// TwinCAT 3 PLC project _2AngleProPLC
// ProgramVersion: 3.1.4024.0
// libraries:
//   Tc2_MC2, * (Beckhoff Automation GmbH)
//   Tc2_Standard, * (Beckhoff Automation GmbH)
//   Tc2_System, * (Beckhoff Automation GmbH)
//   Tc3_Module, * (Beckhoff Automation GmbH)
// project tree:
//   DUTs/ AnalogSignal.TcDUT, SSI_Encoder.TcDUT, ST_IOcard.TcDUT
//   / GlobalTextList.TcGTLO, PlcTask.TcTTO, Visualization Manager.TcVMO (not stored)
//   GVLs/ GVL.TcGVL, GVL_Retain.TcGVL, IO.TcGVL, TwinSAFE.TcGVL
//   POUs/FUNCTION BLOCKS/ FB_AnalogIn.TcPOU, FB_Blinker.TcPOU, FB_IntFilter.TcPOU, FB_SSI_Encoder.TcPOU, InverseAnalogControl.TcPOU
//   POUs/MAIN FUNCTIONS/ PRG_00_General.TcPOU, PRG_01_Reel.TcPOU, PRG_02_Xdrive.TcPOU, PRG_03_Saw.TcPOU, PRG_04_SawAxes.TcPOU, PRG_05_Turret_Carriage.TcPOU, PRG_06_HomePosition.TcPOU, PRG_07_Servo.TcPOU, PRG_08_AnalogSignal.TcPOU, PRG_XX_Visualization_Variables.TcPOU
//   POUs/ MAIN.TcPOU, PRG_IO.TcPOU
//   VISUs/ Visualization.TcVIS
// real-time tasks:
//   TASK PlcTask: cycle T#10ms, priority 20, ADS port 350
// motion (NC):
//   TASK NC-Task 1 SAF: cycle T#2ms, priority 4, ADS port 501
//   TASK NC-Task 1 SVB: cycle T#10ms, priority 8, ADS port 511
//   AXIS Axis 1 (id 1)
//     OtherSettings: AllowMotionCmdToSlave=true
//     encoder EncType=19
//       EncPara: MaxCount=#xffffffff
//     drive DrvType=16
//       DrvPara: MaxCount=#xffffffff, DriveControlDWord=#x00020100
//         Analog: TorqueSetpointScale=10, ScaleFactorActTorque=0.1
//         TimeComp: TaskDelayCycles=1
//     controller CtrType=1
//       CtrPara: PriorControlFactor=1
//         Observer: BandWidth=20
//   AXIS Axis 2 (id 2)
//     OtherSettings: AllowMotionCmdToSlave=true
//     encoder EncType=19
//       EncPara: MaxCount=#xffffffff
//     drive DrvType=16
//       DrvPara: MaxCount=#xffffffff, DriveControlDWord=#x00020100
//         Analog: TorqueSetpointScale=10, ScaleFactorActTorque=0.1
//         TimeComp: TaskDelayCycles=1
//     controller CtrType=1
//       CtrPara: PriorControlFactor=1
//         Observer: BandWidth=20
// I/O:
//   DEVICE Device 1 (EtherCAT), AmsNetId 5.146.75.130.2.1
//     AK1 (EK1200) [EK1200-5000 EtherCAT Power supply (2A E-Bus)]
//       SI1 (EL6910) [EL6910, TwinSAFE PLC]
//       ID1 (EL1018) [EL1018 8Ch. Dig. Input 24V, 10µs]
//       ID2 (EL1018) [EL1018 8Ch. Dig. Input 24V, 10µs]
//       IS1 (EL1904) [EL1904, 4 Ch. Safety Input 24V, TwinSAFE]
//         modules: Module 1 (FSOES)
//       IS2 (EL1904) [EL1904, 4 Ch. Safety Input 24V, TwinSAFE]
//         modules: Module 1 (FSOES)
//       ID3 (EL1018) [EL1018 8Ch. Dig. Input 24V, 10µs]
//       ID4 (EL1018) [EL1018 8Ch. Dig. Input 24V, 10µs]
//       IS3 (EL1904) [EL1904, 4 Ch. Safety Input 24V, TwinSAFE]
//         modules: Module 1 (FSOES)
//       ID5 (EL1018) [EL1018 8Ch. Dig. Input 24V, 10µs]
//       OS1 (EL2904) [EL2904, 4 Ch. Safety Output 24V, 0.5A, TwinSAFE]
//         modules: Module 1 (FSOES), Module 2 (DO)
//       PS1 (EL9410) [EL9410 E-Bus Power Supplier  (Diagnostics)]
//       EN1 (EL5002) [EL5002 2Ch. SSI Encoder]
//       OD1 (EL2008) [EL2008 8Ch. Dig. Output 24V, 0.5A]
//       OD2 (EL2008) [EL2008 8Ch. Dig. Output 24V, 0.5A]
//       OD3 (EL2008) [EL2008 8Ch. Dig. Output 24V, 0.5A]
//       OA1 (EL4104) [EL4104 4Ch. Ana. Output 0-10V, 16bit]
//       IA1 (EL3054) [EL3054 4Ch. Ana. Input 4-20mA]
//       ID6 (EL1018) [EL1018 8Ch. Dig. Input 24V, 10µs]
//       ID7 (EL1018) [EL1018 8Ch. Dig. Input 24V, 10µs]
//       ID8 (EL1018) [EL1018 8Ch. Dig. Input 24V, 10µs]
//       OD4 (EL2008) [EL2008 8Ch. Dig. Output 24V, 0.5A]
//       SD1 (ELM7231-9016) [ELM7231-9016 1Ch. Servo Terminal (48 V, 16 A RMS, OCT, STO, TwinSAFE Logic)]
//         modules: Module 1 (SAFETY)
//       SD2 (ELM7231-9016) [ELM7231-9016 1Ch. Servo Terminal (48 V, 16 A RMS, OCT, STO, TwinSAFE Logic)]
//         modules: Module 1 (SAFETY)
//       ST1 (EL9011) [EL9011 End Terminal]
//   DEVICE Device 4 (COM Port)
// variable links:
//   Device 1 (EtherCAT) <-> Device 1 (EtherCAT)/AK1 (EK1200)/IS1 (EL1904)
//     AK1 (EK1200)/SI1 (EL6910)/ConnectionInputs/Message_5 TxPDO <-> Module 1 (FSOES)/RxPDO/FSOE
//   Device 1 (EtherCAT) <-> Device 1 (EtherCAT)/AK1 (EK1200)/IS3 (EL1904)
//     AK1 (EK1200)/SI1 (EL6910)/ConnectionInputs/Message_7 TxPDO <-> Module 1 (FSOES)/RxPDO/FSOE
//   Device 1 (EtherCAT) <-> Device 1 (EtherCAT)/AK1 (EK1200)/OS1 (EL2904)
//     AK1 (EK1200)/SI1 (EL6910)/ConnectionOutputs/Message_8 RxPDO <-> Module 1 (FSOES)/TxPDO/FSOE
//   Device 1 (EtherCAT) <-> Device 1 (EtherCAT)/AK1 (EK1200)/SD1 (ELM7231-9016)
//     AK1 (EK1200)/SI1 (EL6910)/ConnectionInputs/Message_4 TxPDO <-> Module 1 (SAFETY)/SAFETY FSoE Connection 1 Receive Message/Message_1
//     AK1 (EK1200)/SI1 (EL6910)/ConnectionOutputs/Message_4 RxPDO <-> Module 1 (SAFETY)/SAFETY FSoE Connection 1 Send Message/Message_1
//   Device 1 (EtherCAT) <-> Device 1 (EtherCAT)/AK1 (EK1200)/SD2 (ELM7231-9016)
//     AK1 (EK1200)/SI1 (EL6910)/ConnectionInputs/Message_3 TxPDO <-> Module 1 (SAFETY)/SAFETY FSoE Connection 1 Receive Message/Message_1
//     AK1 (EK1200)/SI1 (EL6910)/ConnectionOutputs/Message_3 RxPDO <-> Module 1 (SAFETY)/SAFETY FSoE Connection 1 Send Message/Message_1
//   Device 1 (EtherCAT) <-> Device 1 (EtherCAT)/AK1 (EK1200)/SI1 (EL6910)
//     AK1 (EK1200)/IS1 (EL1904)/Module 1 (FSOES)/TxPDO/FSOE <-> ConnectionOutputs/Message_5 RxPDO
//     AK1 (EK1200)/IS2 (EL1904)/Module 1 (FSOES)/TxPDO/FSOE <-> ConnectionOutputs/Message_6 RxPDO
//     AK1 (EK1200)/IS3 (EL1904)/Module 1 (FSOES)/TxPDO/FSOE <-> ConnectionOutputs/Message_7 RxPDO
//     AK1 (EK1200)/IS2 (EL1904)/Module 1 (FSOES)/RxPDO/FSOE <-> ConnectionInputs/Message_6 TxPDO
//     AK1 (EK1200)/OS1 (EL2904)/Module 1 (FSOES)/RxPDO/FSOE <-> ConnectionInputs/Message_8 TxPDO
//   NC-Task 1 SAF/Axes/Axis 1 <-> Device 1 (EtherCAT)/AK1 (EK1200)/SD1 (ELM7231-9016)
//     Drive/Inputs/In/nDataIn1 <-> DRV Following error actual value/Following error actual value
//     Drive/Inputs/In/nDcOutputTime <-> InfoData/DcOutputShift
//     Drive/Inputs/In/nState1 <-> DRV Statusword/Statusword
//     Drive/Inputs/In/nState2 <-> DRV Statusword/Statusword @bit 8
//     Drive/Inputs/In/nState4 @bit 1 <-> WcState/InputToggle0
//     Drive/Inputs/In/nState4 <-> WcState/WcState0
//     Drive/Outputs/Out/nCtrl1 <-> DRV Controlword/Controlword
//     Drive/Outputs/Out/nCtrl2 <-> DRV Controlword/Controlword @bit 8
//     Drive/Outputs/Out/nDataOut1 <-> DRV Target position/Target position
//     Enc/Inputs/In/nDataIn1 <-> FB Position/Position
//     Enc/Inputs/In/nDcInputTime <-> InfoData/DcInputShift
//     Enc/Inputs/In/nState4 @bit 1 <-> WcState/InputToggle0
//     Enc/Inputs/In/nState4 <-> WcState/WcState0
//   NC-Task 1 SAF/Axes/Axis 2 <-> Device 1 (EtherCAT)/AK1 (EK1200)/SD2 (ELM7231-9016)
//     Drive/Inputs/In/nDataIn1 <-> DRV Following error actual value/Following error actual value
//     Drive/Inputs/In/nDcOutputTime <-> InfoData/DcOutputShift
//     Drive/Inputs/In/nState1 <-> DRV Statusword/Statusword
//     Drive/Inputs/In/nState2 <-> DRV Statusword/Statusword @bit 8
//     Drive/Inputs/In/nState4 @bit 1 <-> WcState/InputToggle0
//     Drive/Inputs/In/nState4 <-> WcState/WcState0
//     Drive/Outputs/Out/nCtrl1 <-> DRV Controlword/Controlword
//     Drive/Outputs/Out/nCtrl2 <-> DRV Controlword/Controlword @bit 8
//     Drive/Outputs/Out/nDataOut1 <-> DRV Target position/Target position
//     Enc/Inputs/In/nDataIn1 <-> FB Position/Position
//     Enc/Inputs/In/nDcInputTime <-> InfoData/DcInputShift
//     Enc/Inputs/In/nState4 @bit 1 <-> WcState/InputToggle0
//     Enc/Inputs/In/nState4 <-> WcState/WcState0
//   2AngleProPLC/2AngleProPLC Instance <-> Device 1 (EtherCAT)/AK1 (EK1200)/EN1 (EL5002)
//     PlcTask Inputs/IO.IN_uCrossCutSSI <-> SSI Inputs Channel 2/Counter value
//     PlcTask Inputs/IO.IN_uTurretSSI <-> SSI Inputs Channel 1/Counter value
//   2AngleProPLC/2AngleProPLC Instance <-> Device 1 (EtherCAT)/AK1 (EK1200)/IA1 (EL3054)
//     PlcTask Inputs/IO.IN_iCarriagePOSStatus <-> AI Standard Channel 3/Status
//     PlcTask Inputs/IO.IN_iCarriagePOSValue <-> AI Standard Channel 3/Value
//     PlcTask Inputs/IO.IN_iSawCurrentStatus <-> AI Standard Channel 1/Status
//     PlcTask Inputs/IO.IN_iSawCurrentValue <-> AI Standard Channel 1/Value
//   2AngleProPLC/2AngleProPLC Instance <-> Device 1 (EtherCAT)/AK1 (EK1200)/ID1 (EL1018)
//     PlcTask Inputs/IO.ID1/Ch{1..8} <-> Channel {1..8}/Input  (8 links)
//   2AngleProPLC/2AngleProPLC Instance <-> Device 1 (EtherCAT)/AK1 (EK1200)/ID2 (EL1018)
//     PlcTask Inputs/IO.ID2/Ch{1..8} <-> Channel {1..8}/Input  (8 links)
//   2AngleProPLC/2AngleProPLC Instance <-> Device 1 (EtherCAT)/AK1 (EK1200)/ID3 (EL1018)
//     PlcTask Inputs/IO.ID3/Ch{1..8} <-> Channel {1..8}/Input  (8 links)
//   2AngleProPLC/2AngleProPLC Instance <-> Device 1 (EtherCAT)/AK1 (EK1200)/ID4 (EL1018)
//     PlcTask Inputs/IO.ID4/Ch{1..8} <-> Channel {1..8}/Input  (8 links)
//   2AngleProPLC/2AngleProPLC Instance <-> Device 1 (EtherCAT)/AK1 (EK1200)/ID5 (EL1018)
//     PlcTask Inputs/IO.ID5/Ch{1..8} <-> Channel {1..8}/Input  (8 links)
//   2AngleProPLC/2AngleProPLC Instance <-> Device 1 (EtherCAT)/AK1 (EK1200)/ID6 (EL1018)
//     PlcTask Inputs/IO.ID6/Ch{1..8} <-> Channel {1..8}/Input  (8 links)
//   2AngleProPLC/2AngleProPLC Instance <-> Device 1 (EtherCAT)/AK1 (EK1200)/ID7 (EL1018)
//     PlcTask Inputs/IO.ID7/Ch{1..8} <-> Channel {1..8}/Input  (8 links)
//   2AngleProPLC/2AngleProPLC Instance <-> Device 1 (EtherCAT)/AK1 (EK1200)/ID8 (EL1018)
//     PlcTask Inputs/IO.ID8/Ch{1..8} <-> Channel {1..8}/Input  (8 links)
//   2AngleProPLC/2AngleProPLC Instance <-> Device 1 (EtherCAT)/AK1 (EK1200)/OA1 (EL4104)
//     PlcTask Outputs/IO.OUT_iCrossCutFeedback <-> AO Output Channel 2/Analog output
//     PlcTask Outputs/IO.OUT_iEncoderDisplay <-> AO Output Channel 1/Analog output
//   2AngleProPLC/2AngleProPLC Instance <-> Device 1 (EtherCAT)/AK1 (EK1200)/OD1 (EL2008)
//     PlcTask Outputs/IO.OD1/Ch{1..8} <-> Channel {1..8}/Output  (8 links)
//   2AngleProPLC/2AngleProPLC Instance <-> Device 1 (EtherCAT)/AK1 (EK1200)/OD2 (EL2008)
//     PlcTask Outputs/IO.OD2/Ch{1..8} <-> Channel {1..8}/Output  (8 links)
//   2AngleProPLC/2AngleProPLC Instance <-> Device 1 (EtherCAT)/AK1 (EK1200)/OD3 (EL2008)
//     PlcTask Outputs/IO.OD3/Ch{1..8} <-> Channel {1..8}/Output  (8 links)
//   2AngleProPLC/2AngleProPLC Instance <-> Device 1 (EtherCAT)/AK1 (EK1200)/OD4 (EL2008)
//     PlcTask Outputs/IO.OD4/Ch{1..8} <-> Channel {1..8}/Output  (8 links)
//   2AngleProPLC/2AngleProPLC Instance <-> Device 1 (EtherCAT)/AK1 (EK1200)/SD1 (ELM7231-9016)
//     PlcTask Outputs/TwinSAFE.SafeErrAck <-> Module 1 (SAFETY)/SAFETY Standard Outputdata/Standard In Var 3
//     PlcTask Outputs/TwinSAFE.SafeRUN <-> Module 1 (SAFETY)/SAFETY Standard Outputdata/Standard In Var 2
//   2AngleProPLC/2AngleProPLC Instance <-> Device 1 (EtherCAT)/AK1 (EK1200)/SD2 (ELM7231-9016)
//     PlcTask Outputs/TwinSAFE.SafeErrAck <-> Module 1 (SAFETY)/SAFETY Standard Outputdata/Standard In Var 3
//     PlcTask Outputs/TwinSAFE.SafeRUN <-> Module 1 (SAFETY)/SAFETY Standard Outputdata/Standard In Var 2
//   2AngleProPLC/2AngleProPLC Instance <-> Device 1 (EtherCAT)/AK1 (EK1200)/SI1 (EL6910)
//     PlcTask Inputs/TwinSAFE.IN_FaultReset <-> StandardInputs/Standard Out Var 9
//     PlcTask Inputs/TwinSAFE.OUT_STO <-> StandardInputs/Standard Out Var 10
//     PlcTask Outputs/TwinSAFE.SafeErrAck <-> StandardOutputs/Standard In Var 2
//     PlcTask Outputs/TwinSAFE.SafeRUN <-> StandardOutputs/Standard In Var 1
//   2AngleProPLC/2AngleProPLC Instance <-> NC-Task 1 SAF/Axes/Axis 1
//     PlcTask Inputs/GVL.Ax1.NcToPlc <-> Outputs/ToPlc
//     PlcTask Outputs/GVL.Ax1.PlcToNc <-> Inputs/FromPlc
//   2AngleProPLC/2AngleProPLC Instance <-> NC-Task 1 SAF/Axes/Axis 2
//     PlcTask Inputs/GVL.Ax2.NcToPlc <-> Outputs/ToPlc
//     PlcTask Outputs/GVL.Ax2.PlcToNc <-> Inputs/FromPlc

CONFIGURATION _2AngleProPLC
    RESOURCE PLC ON TwinCAT3
        TASK PlcTask(INTERVAL := T#10ms, PRIORITY := 20);
        PROGRAM MAIN WITH PlcTask : MAIN;
    END_RESOURCE
END_CONFIGURATION

// ---- DUTs/AnalogSignal.TcDUT
TYPE AnalogSignal :
STRUCT
	iRawVal 		: INT; 	(* raw readout *)
	rScaled 		: REAL; (* scaled value between min and max *)
	bUnderRange 	: BOOL;
	bOverRange 		: BOOL;
	bLimit1			: BYTE;
	bLimit2			: BYTE;
	bError			: BOOL;
	bPDO_State		: BOOL;
	bPDO_Toggle		: BOOL;
END_STRUCT
END_TYPE

// ---- DUTs/SSI_Encoder.TcDUT
TYPE SSI_Encoder :
STRUCT
	uCounterValue	: UDINT ;		// Raw counter value
	rScaled			: REAL ;		// scaled value
	bDataError		: BOOL ;		
	bFrameError		: BOOL ;
	bPowerFailure	: BOOL ;
	bDataMismatch	: BOOL ;
	bSyncError		: BOOL ;
	bPDO_State		: BOOL ;
	bPDO_Toggle		: BOOL ;
END_STRUCT
END_TYPE

// ---- DUTs/ST_IOcard.TcDUT
TYPE ST_IOcard :
STRUCT
	Ch1	:	BOOL;
	Ch2	:	BOOL;
	Ch3	:	BOOL;
	Ch4	:	BOOL;
	Ch5	:	BOOL;
	Ch6	:	BOOL;
	Ch7	:	BOOL;
	Ch8	:	BOOL;
END_STRUCT
END_TYPE

// ---- GVLs/GVL.TcGVL
VAR_GLOBAL
	
	bSafetyOK		: BOOL ;
	bAutoCrossCut	: BOOL ;
	bMachineHoming: BOOL;
	bTurretHome: BOOL;
	bCarriageHomeRH: BOOL;
	bCarriageHomeLH: BOOL;
	bCrossCutHomeLH: BOOL;
	bCrossCutHomeRH: BOOL;
	bZAxisHome: BOOL;
	
	fbTurretSSI: FB_SSI_Encoder;
	fbCrossCutSSI: FB_SSI_Encoder;
	fbSawCurrent: FB_AnalogIn;
	fbCarriagePOS: FB_AnalogIn;
	
	bLimitLeft: BOOL;
    bLimitRight: BOOL;
	bCrossCutCentre: BOOL;
	bCrossCutCentreForRotation: BOOL;
	bApproachingLimitRight: BOOL;
	bApproachingLimitLeft: BOOL;
	uCrossCutMedian: UDINT;
	
	bTurretReturn: BOOL;
	TurretReturn: SR;
	bTriggerReset: BOOL;
	bTurretMedianRange: BOOL;
	bTurretBufferSpeed: BOOL;
	
	Ax1	:	AXIS_REF;
	Ax2	:	AXIS_REF;
	fbMC_GearIn: MC_GearIn;
	
	bSawUP		:	BOOL;
	bSawDOWN	:	BOOL;
	
	bAnyServoError: BOOL;
	bAutoCrossCutErr: BOOL;
	
	uTurretSSIMedian: UDINT;
	bTurretUnderMedian: BOOL;
	bTurretOverMedian: BOOL;
	bTurret045Range: BOOL;
	
	RS_TriggerStopLH: RS;
	RS_TriggerStopRH: RS;
	
	fbCarriageValueFilter: FB_IntFilter;
	rCrossCutSpeedMultiplier: REAL;
	uRailLimitLeft: UDINT;
	uRailLimitRight: UDINT;
	bEchainCrashPosLeft: BOOL;
	bEchainCrashPosRight: BOOL;
	
	bTurretMedian: BOOL;
	bTurretCW: BOOL;
	bTurretCCW: BOOL;
	
	// Visualization Variables
	bRemote: BOOL;
	bAutoCrossCutSingle: BOOL;
	bAutoCrossCutDouble: BOOL;
	bZAxisSlow: BOOL;
	bZAxisMed: BOOL;
	bZAxisFast: BOOL;
	bTrtCCW: BOOL;
	bTrtCW: BOOL;
	bCrgLH: BOOL;
	bCrgRH: BOOL;
	bTeachLeft: BOOL;
	bTeachRight: BOOL;
END_VAR

// ---- GVLs/GVL_Retain.TcGVL
VAR_GLOBAL RETAIN

	uTeachLimitLeft: UDINT;
	uTeachLimitRight: UDINT;
	iCarriageMedian: INT;
	iCarriageLeftLimit: INT;
	iCarriageRightLimit: INT;
	iZAxisUpperLimitValue: DINT;
	iZAxisLowerLimitValue: DINT;
	uTRTCaptureValueMin: UDINT;
    uTRTCaptureValueMax: UDINT;
END_VAR

// ---- GVLs/IO.TcGVL
VAR_GLOBAL
	
	ID1							AT%I*		: ST_IOcard ;
	ID2							AT%I*		: ST_IOcard ;
	ID3							AT%I*		: ST_IOcard ;
	ID4							AT%I*		: ST_IOcard ;
	ID5							AT%I*		: ST_IOcard ;
	ID6							AT%I*		: ST_IOcard ;
	ID7							AT%I*		: ST_IOcard ;	
	ID8							AT%I*		: ST_IOcard ;	
	
	IN_iSawCurrentValue			AT%IW100	: INT ;
	IN_iSawCurrentStatus		AT%IW101	: INT ;
	
//	IN_iDrvFeedbackValue		AT%IW130	: INT ;
//	IN_iDrvFeedbackStatus		AT%IW131	: INT ;
	
	IN_iCarriagePOSValue		AT%IW136	: INT ;
	IN_iCarriagePOSStatus		AT%IW137	: INT ;
	
//	IN_iCarriageTESTValue		AT%IW140	: INT ;
//	IN_iCarriageTESTStatus		AT%IW141 	: INT ;

	OD1							AT%Q*		: ST_IOcard ;
	OD2							AT%Q*		: ST_IOcard ;
	OD3							AT%Q*		: ST_IOcard ;
	OD4							AT%Q*		: ST_IOcard ;
	
	OUT_iEncoderDisplay			AT%QW105	: INT ;
	OUT_iCrossCutFeedback		AT%QW106	: INT ;
//	OUT_iXDriveFeedback			AT%QW107	: INT ;

	
	IN_uTurretSSI				AT%IW110	: UDINT ;
	IN_uCrossCutSSI				AT%IW116	: UDINT ;

	
	
			(* INPUTS *)
// ID1			
	IN_bSawON					: BOOL;
	IN_bTeach					: BOOL;
	IN_bSprayer					: BOOL;
	IN_bRemote					: BOOL;
	IN_bCableReel				: BOOL;
	IN_bHoseReel				: BOOL;
	IN_bWaterLine				: BOOL;
	IN_bFieldLight				: BOOL;
	
// ID2	                    		
	IN_bTeachLeft				: BOOL;
	IN_bTeachRight				: BOOL;
	IN_bSawReturnLimit			: BOOL;
// IN_b						: BOOL;
	IN_bSawUpLimit				: BOOL;
	IN_bSawDownLimit			: BOOL;
	IN_bDoublePassReference		: BOOL;
//	IN_b						: BOOL;

// ID3	                    		
	IN_bSawUP					: BOOL;
	IN_bSawDOWN					: BOOL;
	IN_bSawCUT					: BOOL;
	IN_bSawRETURN				: BOOL;
	IN_bCarriageLH				: BOOL;
	IN_bCarriageRH				: BOOL;
	IN_bXDriveFwd				: BOOL;
	IN_bXDriveRev				: BOOL;

// ID4	                        	
	IN_bCrossCutLeft			: BOOL;
	IN_bCrossCutRight			: BOOL;
	IN_bLiftingPosition			: BOOL;
	IN_bHorn					: BOOL;
	IN_bTrtCrgReady				: BOOL;
	IN_bDriveReady				: BOOL;
	IN_bCrossCutReady			: BOOL;
	IN_bSawMOLReady				: BOOL;

// ID5	                        	
	IN_bCableReelMOLReady		: BOOL;
	IN_bHoseReelMOLReady		: BOOL;
	IN_b48VDCReady				: BOOL;
	IN_bCrgMOLReady				: BOOL;
	IN_bTrtMOLReady				: BOOL;
	IN_bZaxisSlow				: BOOL;
	IN_bZaxisFast				: BOOL;
//	IN_b						: BOOL;

// ID6	
	IN_bRemoteUP            	: BOOL;
	IN_bRemoteDOWN				: BOOL;
	IN_bRemoteCUT    			: BOOL;
	IN_bRemoteRETURN			: BOOL;
	IN_bRemoteCrgLH   			: BOOL;
	IN_bRemoteCrgRH				: BOOL;
	IN_bRemoteTrtCCW 			: BOOL;
	IN_bRemoteTrtCW				: BOOL;	

// ID7	
	IN_bRemoteDrvFwd			: BOOL;
	IN_bRemoteDrvRev			: BOOL;
	IN_bRemoteSawON				: BOOL;
	IN_bRemoteStop				: BOOL;
	IN_bTurretCW				: BOOL;
	IN_bTurretCCW				: BOOL;
	IN_bTurretReturn			: BOOL;
	IN_bAutoCrossCutDouble		: BOOL;

// ID8	
	IN_bTurretReference  		: BOOL;
	IN_bTurretCWLimit    		: BOOL;
	IN_bTurretCCWLimit	    	: BOOL;
//	IN_b					    : BOOL;
	IN_bCarriageLHLimit			: BOOL;
	IN_bCarriageRHLimit			: BOOL;
	IN_bCarriageReference		: BOOL;
	IN_bTurretRotationReference	: BOOL;
	                        	
			(* OUTPUTS *) 
// OD1  	
	OUT_bCrgContactor			: BOOL;
	OUT_bTrtContactor			: BOOL;
	OUT_bTrtCrgLH				: BOOL;
	OUT_bTrtCrgRH				: BOOL;
	OUT_bTurretSpeed			: BOOL;
	OUT_bCarriageSpeed			: BOOL;
	OUT_bSawCUT					: BOOL;
	OUT_bSawRETURN				: BOOL;

// OD2	                        	
	OUT_bXDriveFwd				: BOOL;
	OUT_bXDriveRev				: BOOL;
	OUT_bSawON					: BOOL;
	OUT_bCableReel				: BOOL;
	OUT_bHoseReel				: BOOL;
	OUT_bFaultResetLED			: BOOL;
	OUT_bSawONLED				: BOOL;
	OUT_bRipCutSpeed			: BOOL;

// OD3	                        	
	OUT_bTravelSpeedLED			: BOOL; 
	OUT_bTurretReturnLED		: BOOL;
	OUT_bFieldLight				: BOOL;
	OUT_bSprayer				: BOOL;
	OUT_bSignalLightReelside	: BOOL;
	OUT_bSignalLightPanelside	: BOOL;
	OUT_bHorn					: BOOL;
	OUT_bWaterLine				: BOOL; 

// OD4	
	OUT_bTeachLED				: BOOL;
	OUT_bLiftingPositionLED		: BOOL;
	OUT_bCarriageReferenceLED	: BOOL;
	OUT_bTurretReferenceLED		: BOOL;
//	OUT_b						: BOOL;
//	OUT_b						: BOOL;
//	OUT_b						: BOOL;
//	OUT_b						: BOOL;
	

END_VAR

// ---- GVLs/TwinSAFE.TcGVL
VAR_GLOBAL
	SafeRUN		AT%Q*	: BOOL := TRUE ;
	SafeErrAck	AT%Q*	: BOOL ;
	
		
	IN_FaultReset	AT%I*	: BOOL ;
	IN_EDM			AT%I*	: BOOL ;
	OUT_STO			AT%I*	: BOOL ;
	
END_VAR

// ---- POUs/MAIN.TcPOU
PROGRAM MAIN
VAR
	FB_Blinker_TrtCrgReferenceLED: FB_Blinker;
END_VAR

PRG_IO();

PRG_00_General();
PRG_01_Reel();
PRG_02_Xdrive();
PRG_03_Saw();
PRG_04_SawAxes();
	PRG_04_SawAxes.ACT_04_1_AutoCrossCut();
	PRG_04_SawAxes.ACT_04_2_CrossCutSpeed();	// CURRENT FEEDBACK
PRG_05_Turret_Carriage();
PRG_06_HomePosition();
PRG_07_Servo();
	PRG_07_Servo.ACT_07_1_Power();
	PRG_07_Servo.ACT_07_2_Reset();
	PRG_07_Servo.ACT_07_3_Jog();
	PRG_07_Servo.ACT_07_4_JogSpeed();
	PRG_07_Servo.ACT_07_5_Stop();
PRG_08_AnalogSignal();
	PRG_08_AnalogSignal.ACT_08_1_TurretSSI();
	PRG_08_AnalogSignal.ACT_08_2_CrossCutSSI();
	PRG_08_AnalogSignal.ACT_08_3_CarriagePOS();
PRG_XX_Visualization_Variables();

SafeErrAck := IN_FaultReset ;

	// Outputs unaffected by Safety system
OUT_bFieldLight		:= IN_bFieldLight	;
OUT_bSprayer := IN_bSprayer ;
		FB_Blinker_TrtCrgReferenceLED(IN:= TRUE, blink_time:= T#0.5S, OUT=> );

	IF bTurretMedianRange THEN
		OUT_bTurretReferenceLED := TRUE ;
	ELSIF (bCrossCutCentreForRotation AND NOT IN_bCarriageReference) THEN
		OUT_bTurretReferenceLED := FB_Blinker_TrtCrgReferenceLED.OUT ;
	ELSE OUT_bTurretReferenceLED := FALSE ;
	END_IF
	
	IF NOT IN_bCarriageReference THEN 
		OUT_bCarriageReferenceLED := TRUE ;
	ELSIF fbCrosscutSSI.Out.rScaled <= (((fbCrosscutSSI.MaxOut - fbCrosscutSSI.MinOut)/2)+12) AND fbCrosscutSSI.Out.rScaled >= (((fbCrosscutSSI.MaxOut - fbCrosscutSSI.MinOut)/2)-12) THEN
		OUT_bCarriageReferenceLED := FB_Blinker_TrtCrgReferenceLED.OUT ;
	ELSE OUT_bCarriageReferenceLED := FALSE ;
	END_IF

END_PROGRAM

// ---- POUs/FUNCTION BLOCKS/FB_Blinker.TcPOU
FUNCTION_BLOCK FB_Blinker
VAR_INPUT
	IN			:	BOOL;
	blink_time	:	TIME;
END_VAR
VAR_OUTPUT
	OUT			:	BOOL;
END_VAR
VAR
	timerON		:	TON;
	timerOFF	:	TOF;
END_VAR

timerON(IN:= 	IN AND NOT timerOFF.Q,
		PT:=	blink_time , 
		Q=>		, 
		ET=> );

timerOFF(IN:= 	timerON.Q ,
		PT:=	blink_time , 
		Q=> 	OUT, 
		ET=> );

END_FUNCTION_BLOCK

// ---- POUs/PRG_IO.TcPOU
PROGRAM PRG_IO
VAR
END_VAR

			(* INPUTS *)
	IN_bSawON		    		:= IO.ID1.Ch1 ;
	IN_bTeach		     		:= IO.ID1.Ch2 ;
	IN_bSprayer	  				:= IO.ID1.Ch3 ;
	IN_bRemote		 			:= IO.ID1.Ch4 ;
	IN_bCableReel	 			:= IO.ID1.Ch5 ;
	IN_bHoseReel	  			:= IO.ID1.Ch6 ;
	IN_bWaterLine	 			:= IO.ID1.Ch7 ;
	IN_bFieldLight				:= IO.ID1.Ch8 ;
	                    	  
	IN_bTeachLeft			    := IO.ID2.Ch1 ;
	IN_bTeachRight			    := IO.ID2.Ch2 ;
	IN_bSawReturnLimit		   	:= IO.ID2.Ch3 ;
//	IN_b					    := IO.ID2.Ch4 ;
	IN_bSawUpLimit			    := IO.ID2.Ch5 ;
	IN_bSawDownLimit		   	:= IO.ID2.Ch6 ;
	IN_bDoublePassReference		:= IO.ID2.Ch7 ;
//	IN_b					    := IO.ID2.Ch8 ;
	                    	  
	IN_bSawUP		    		:= IO.ID3.Ch1 ;
	IN_bSawDOWN		  			:= IO.ID3.Ch2 ;
	IN_bSawCUT		  		 	:= IO.ID3.Ch3 ;
	IN_bSawRETURN	 			:= IO.ID3.Ch4 ;
	IN_bCarriageLH				:= IO.ID3.Ch5 ;
	IN_bCarriageRH				:= IO.ID3.Ch6 ;
	IN_bXDriveFwd	 			:= IO.ID3.Ch7 ;
	IN_bXDriveRev		 		:= IO.ID3.Ch8 ;
	                          
	IN_bCrossCutLeft	        := IO.ID4.Ch1 ;
	IN_bCrossCutRight	        := IO.ID4.Ch2 ;
	IN_bLiftingPosition			:= IO.ID4.Ch3 ;	
	IN_bHorn					:= IO.ID4.Ch4 ;	
	IN_bTrtCrgReady		 		:= IO.ID4.Ch5 ; 
	IN_bDriveReady		  		:= IO.ID4.Ch6 ;	
	IN_bCrossCutReady			:= IO.ID4.Ch7 ;	
	IN_bSawMOLReady		 		:= IO.ID4.Ch8 ;	
	
	IN_bCableReelMOLReady		:= IO.ID5.Ch1 ;
	IN_bHoseReelMOLReady	    := IO.ID5.Ch2 ;
	IN_b48VDCReady			    := IO.ID5.Ch3 ;
	IN_bCrgMOLReady			    := IO.ID5.Ch4 ;
	IN_bTrtMOLReady			    := IO.ID5.Ch5 ;
	IN_bZaxisSlow				:= IO.ID5.Ch6 ;
	IN_bZaxisFast				:= IO.ID5.Ch7 ;
	IN_bTurretRotationReference	:= IO.ID5.Ch8 ;
	
	IN_bRemoteUP            	:= IO.ID6.Ch1 ;
	IN_bRemoteDOWN			    := IO.ID6.Ch2 ;
	IN_bRemoteCUT    		    := IO.ID6.Ch3 ;
	IN_bRemoteRETURN		    := IO.ID6.Ch4 ;
	IN_bRemoteCrgLH   		    := IO.ID6.Ch5 ;
	IN_bRemoteCrgRH			    := IO.ID6.Ch6 ;
	IN_bRemoteTrtCCW 		    := IO.ID6.Ch7 ;
	IN_bRemoteTrtCW			    := IO.ID6.Ch8 ;	
	                        
	IN_bRemoteDrvFwd		   	:= IO.ID7.Ch1 ;
	IN_bRemoteDrvRev		   	:= IO.ID7.Ch2 ;
	IN_bRemoteSawON				:= IO.ID7.Ch3 ;
	IN_bRemoteStop		    	:= IO.ID7.Ch4 ;	
	IN_bTurretCW				:= IO.ID7.Ch5 ;
	IN_bTurretCCW				:= IO.ID7.Ch6 ;
	IN_bTurretReturn		   	:= IO.ID7.Ch7 ;
	IN_bAutoCrossCutDouble	 	:= IO.ID7.Ch8 ;

	
	IN_bTurretReference  	  	:= IO.ID8.Ch1 ;
	IN_bTurretCWLimit    	   	:= IO.ID8.Ch2 ;
	IN_bTurretCCWLimit	     	:= IO.ID8.Ch3 ;
//	IN_b					    := IO.ID8.Ch4 ;
	IN_bCarriageLHLimit		  	:= IO.ID8.Ch5 ;
	IN_bCarriageRHLimit		  	:= IO.ID8.Ch6 ;
	IN_bCarriageReference	 	:= IO.ID8.Ch7 ;
	IN_bTurretRotationReference	:= IO.ID8.Ch8 ;
	
			(* OUTPUTS *)
	IO.OD1.Ch1					:=	OUT_bCrgContactor		;
	IO.OD1.Ch2					:=	OUT_bTrtContactor		;
	IO.OD1.Ch4					:=	OUT_bTrtCrgLH		   	;
	IO.OD1.Ch3					:=	OUT_bTrtCrgRH		   	;
	IO.OD1.Ch5					:=	OUT_bTurretSpeed	    ;
	IO.OD1.Ch6					:=	OUT_bCarriageSpeed	  	;
	IO.OD1.Ch7					:=	OUT_bSawCUT			  	;
	IO.OD1.Ch8					:=	OUT_bSawRETURN		  	;
	            			
	IO.OD2.Ch1					:=	OUT_bXDriveFwd		   	;
	IO.OD2.Ch2					:=	OUT_bXDriveRev		   	;
	IO.OD2.Ch3					:=	OUT_bSawON		    	;
	IO.OD2.Ch4					:=	OUT_bCableReel		   	;
	IO.OD2.Ch5					:=	OUT_bHoseReel		   	;
	IO.OD2.Ch6					:=	OUT_bFaultResetLED		;
	IO.OD2.Ch7					:=	OUT_bSawONLED	    	;
	IO.OD2.Ch8					:=	OUT_bRipCutSpeed	  	;
	            			
	IO.OD3.Ch1					:=	OUT_bTravelSpeedLED		;
	IO.OD3.Ch2					:=	OUT_bTurretReturnLED	;
	IO.OD3.Ch3					:=	OUT_bFieldLight			;
	IO.OD3.Ch4					:=	OUT_bSprayer     		;
	IO.OD3.Ch5					:=	OUT_bSignalLightReelside;	
	IO.OD3.Ch6					:=	OUT_bSignalLightPanelside;	
	IO.OD3.Ch7					:=	OUT_bHorn			    ;	
	IO.OD3.Ch8					:=	OUT_bWaterLine		    ;
	
	IO.OD4.Ch1					:=	OUT_bTeachLED			;
	IO.OD4.Ch2					:=	OUT_bLiftingPositionLED ;
	IO.OD4.Ch3					:=	OUT_bCarriageReferenceLED;
	IO.OD4.Ch4					:=	OUT_bTurretReferenceLED ;
//	IO.OD4.Ch5					:=	OUT_b                   ;
//	IO.OD4.Ch6					:=	OUT_b                   ;
//	IO.OD4.Ch7					:=	OUT_b                   ;
//	IO.OD4.Ch8					:=	OUT_b                   ;

END_PROGRAM

// ---- POUs/MAIN FUNCTIONS/PRG_00_General.TcPOU
PROGRAM PRG_00_General
VAR
	sr_Fault: SR;
	FB_Blinker_ServoError: FB_Blinker;
END_VAR

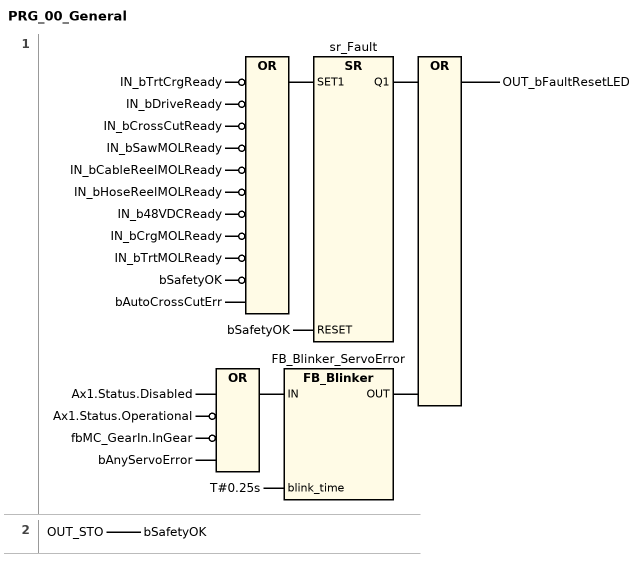
// NETWORK 1
sr_Fault(SET1 := NOT IN_bTrtCrgReady OR NOT IN_bDriveReady OR NOT IN_bCrossCutReady OR NOT IN_bSawMOLReady OR NOT IN_bCableReelMOLReady OR NOT IN_bHoseReelMOLReady OR NOT IN_b48VDCReady OR NOT IN_bCrgMOLReady OR NOT IN_bTrtMOLReady OR NOT bSafetyOK OR bAutoCrossCutErr, RESET := bSafetyOK); // SR
FB_Blinker_ServoError(IN := Ax1.Status.Disabled OR NOT Ax1.Status.Operational OR NOT fbMC_GearIn.InGear OR bAnyServoError, blink_time := T#0.25s); // FB_Blinker
OUT_bFaultResetLED := sr_Fault.Q1 OR FB_Blinker_ServoError.OUT;

// NETWORK 2
bSafetyOK := OUT_STO;

END_PROGRAM

// ---- POUs/MAIN FUNCTIONS/PRG_01_Reel.TcPOU
PROGRAM PRG_01_Reel
VAR
END_VAR

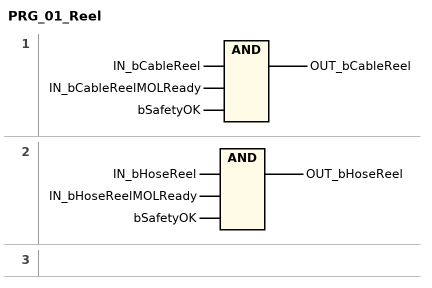
// NETWORK 1
OUT_bCableReel := IN_bCableReel AND IN_bCableReelMOLReady AND bSafetyOK;

// NETWORK 2
OUT_bHoseReel := IN_bHoseReel AND IN_bHoseReelMOLReady AND bSafetyOK;

// NETWORK 3

END_PROGRAM

// ---- POUs/MAIN FUNCTIONS/PRG_02_Xdrive.TcPOU
PROGRAM PRG_02_Xdrive
VAR
	TOF_horn: TOF;
	bRipCut: BOOL;
	signal_light_blink_fwd: FB_Blinker;
	signal_light_blink_rev: FB_Blinker;
	signal_light_blink1: FB_Blinker;
	signal_light_blink2: FB_Blinker;
	R_TRIG_2: R_TRIG;
	R_TRIG_3: R_TRIG;
	bRemoteDRV :BOOL;
	bRemoteREV :BOOL;
	TOF_0: TOF;
	TOF_1: TOF;
	F_TRIG_0: F_TRIG;
	F_TRIG_1: F_TRIG;
END_VAR
VAR // added by the converter: edge detectors and wires of the graphical bodies
    _w1, _w2 : BOOL;
END_VAR

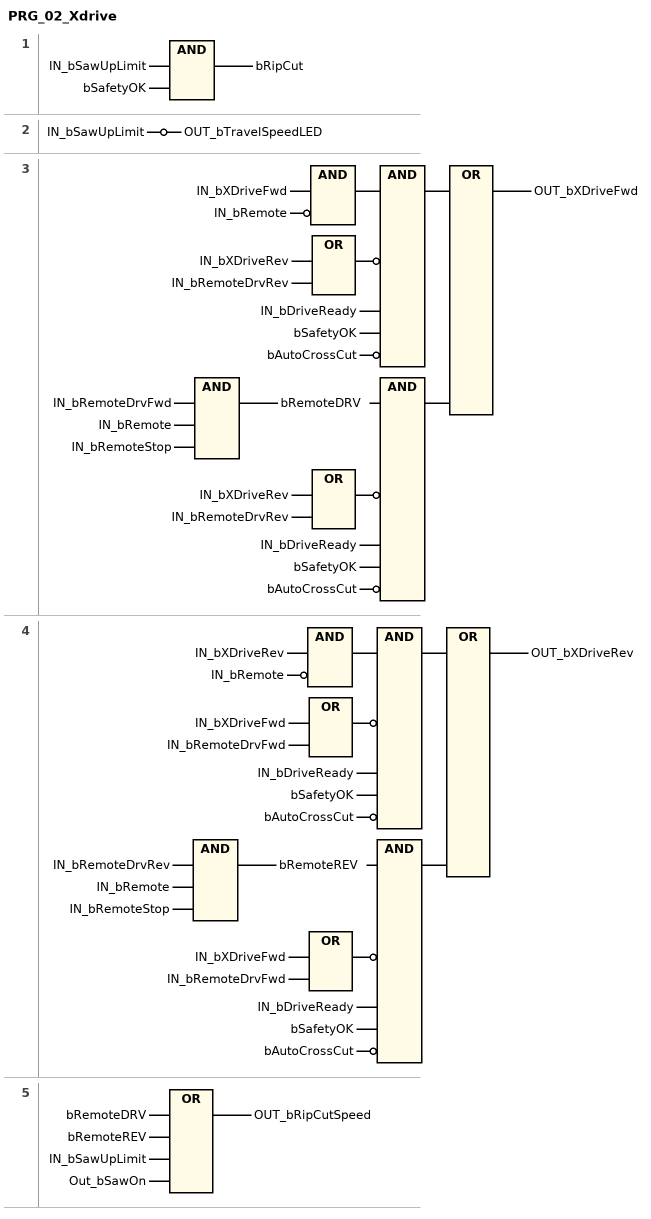
// NETWORK 1
bRipCut := IN_bSawUpLimit AND bSafetyOK;

// NETWORK 2
OUT_bTravelSpeedLED := NOT IN_bSawUpLimit;

// NETWORK 3
_w1 := IN_bRemoteDrvFwd AND IN_bRemote AND IN_bRemoteStop;
bRemoteDRV := _w1;
OUT_bXDriveFwd := (IN_bXDriveFwd AND NOT IN_bRemote) AND NOT (IN_bXDriveRev OR IN_bRemoteDrvRev) AND IN_bDriveReady AND bSafetyOK AND NOT bAutoCrossCut OR _w1 AND NOT (IN_bXDriveRev OR IN_bRemoteDrvRev) AND IN_bDriveReady AND bSafetyOK AND NOT bAutoCrossCut;

// NETWORK 4
_w2 := IN_bRemoteDrvRev AND IN_bRemote AND IN_bRemoteStop;
bRemoteREV := _w2;
OUT_bXDriveRev := (IN_bXDriveRev AND NOT IN_bRemote) AND NOT (IN_bXDriveFwd OR IN_bRemoteDrvFwd) AND IN_bDriveReady AND bSafetyOK AND NOT bAutoCrossCut OR _w2 AND NOT (IN_bXDriveFwd OR IN_bRemoteDrvFwd) AND IN_bDriveReady AND bSafetyOK AND NOT bAutoCrossCut;

// NETWORK 5
OUT_bRipCutSpeed := bRemoteDRV OR bRemoteREV OR IN_bSawUpLimit OR Out_bSawOn;

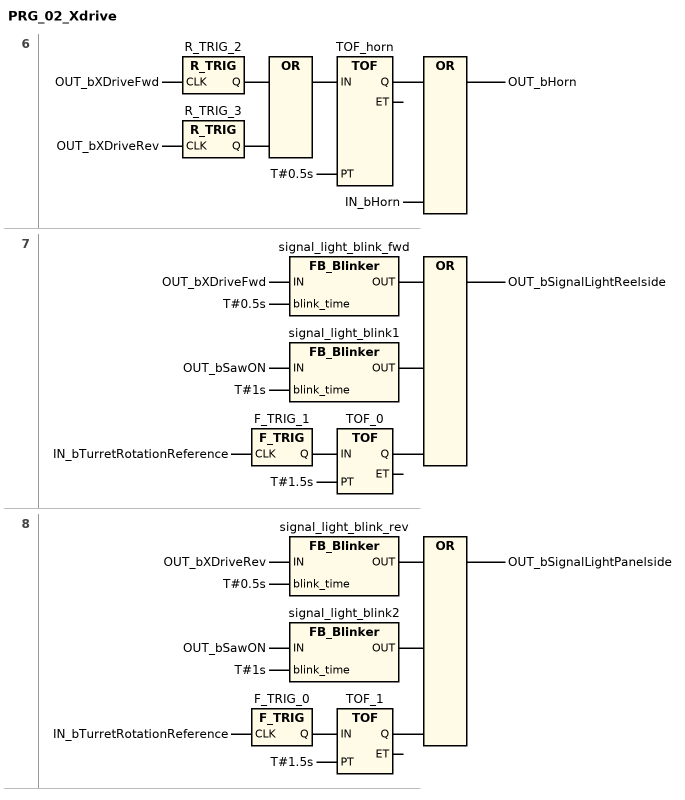
// NETWORK 6
R_TRIG_2(CLK := OUT_bXDriveFwd); // R_TRIG
R_TRIG_3(CLK := OUT_bXDriveRev); // R_TRIG
TOF_horn(IN := R_TRIG_2.Q OR R_TRIG_3.Q, PT := T#0.5s); // TOF
OUT_bHorn := TOF_horn.Q OR IN_bHorn;

// NETWORK 7
signal_light_blink_fwd(IN := OUT_bXDriveFwd, blink_time := T#0.5s); // FB_Blinker
signal_light_blink1(IN := OUT_bSawON, blink_time := T#1s); // FB_Blinker
F_TRIG_1(CLK := IN_bTurretRotationReference); // F_TRIG
TOF_0(IN := F_TRIG_1.Q, PT := T#1.5s); // TOF
OUT_bSignalLightReelside := signal_light_blink_fwd.OUT OR signal_light_blink1.OUT OR TOF_0.Q;

// NETWORK 8
signal_light_blink_rev(IN := OUT_bXDriveRev, blink_time := T#0.5s); // FB_Blinker
signal_light_blink2(IN := OUT_bSawON, blink_time := T#1s); // FB_Blinker
F_TRIG_0(CLK := IN_bTurretRotationReference); // F_TRIG
TOF_1(IN := F_TRIG_0.Q, PT := T#1.5s); // TOF
OUT_bSignalLightPanelside := signal_light_blink_rev.OUT OR signal_light_blink2.OUT OR TOF_1.Q;

END_PROGRAM

// ---- POUs/MAIN FUNCTIONS/PRG_03_Saw.TcPOU
PROGRAM PRG_03_Saw
VAR
	b_SRout: BOOL;	
	SR_saw: SR;
	R_TRIG_0: R_TRIG;
	R_TRIG_1: R_TRIG;
	R_TRIG_3: R_TRIG;
	R_TRIG_2: R_TRIG;
	R_TRIG_4: R_TRIG;
END_VAR
VAR // added by the converter: edge detectors and wires of the graphical bodies
    _w1 : BOOL;
END_VAR

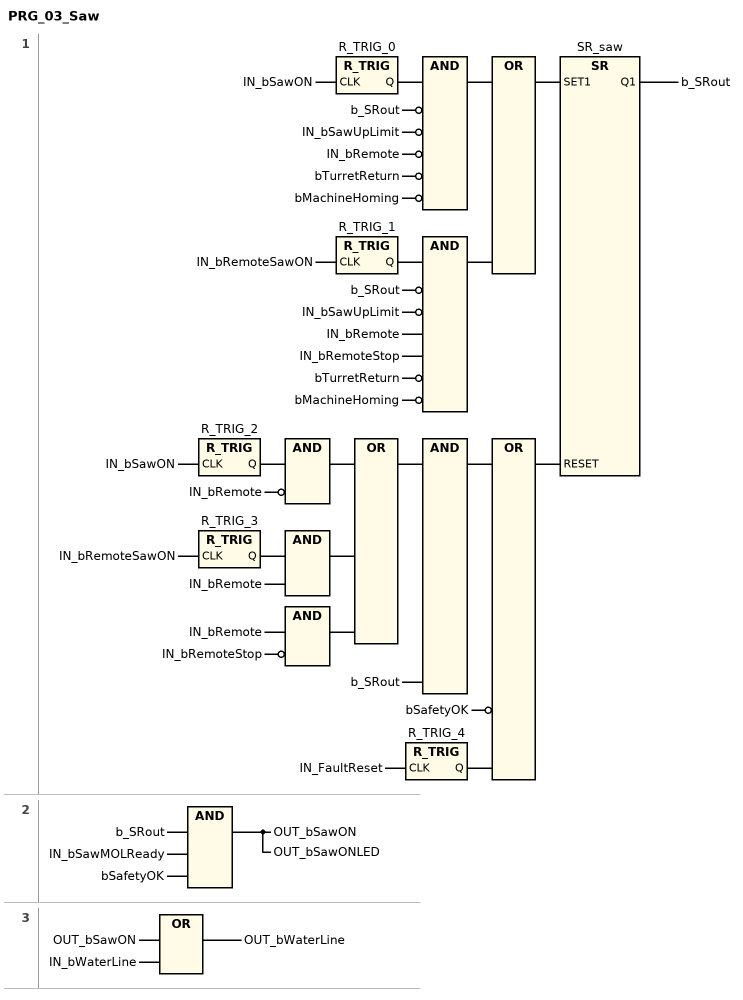
// NETWORK 1
R_TRIG_0(CLK := IN_bSawON); // R_TRIG
R_TRIG_1(CLK := IN_bRemoteSawON); // R_TRIG
R_TRIG_2(CLK := IN_bSawON); // R_TRIG
R_TRIG_3(CLK := IN_bRemoteSawON); // R_TRIG
R_TRIG_4(CLK := IN_FaultReset); // R_TRIG
SR_saw(SET1 := R_TRIG_0.Q AND NOT b_SRout AND NOT IN_bSawUpLimit AND NOT IN_bRemote AND NOT bTurretReturn AND NOT bMachineHoming OR R_TRIG_1.Q AND NOT b_SRout AND NOT IN_bSawUpLimit AND IN_bRemote AND IN_bRemoteStop AND NOT bTurretReturn AND NOT bMachineHoming, RESET := (R_TRIG_2.Q AND NOT IN_bRemote OR R_TRIG_3.Q AND IN_bRemote OR IN_bRemote AND NOT IN_bRemoteStop) AND b_SRout OR NOT bSafetyOK OR R_TRIG_4.Q); // SR
b_SRout := SR_saw.Q1;

// NETWORK 2
_w1 := b_SRout AND IN_bSawMOLReady AND bSafetyOK;
OUT_bSawON := _w1;
OUT_bSawONLED := _w1;

// NETWORK 3
OUT_bWaterLine := OUT_bSawON OR IN_bWaterLine;

END_PROGRAM

// ---- POUs/MAIN FUNCTIONS/PRG_04_SawAxes.TcPOU
PROGRAM PRG_04_SawAxes
VAR
	bUP						: BOOL;
	bDOWN					: BOOL;
	bCUT					: BOOL;
	bRETURN					: BOOL;
	
	bDoublePassCountUp		: BOOL;
	
	ctu_DoublePass			: CTU;
	
	iStep: INT;
	bUP_TON: TON;
//	bUP_TP: TP;
	rtrig1: r_trig;
//	ftrig1: f_trig;
	DoublePass_SR: SR;
	bDoublePassQ: BOOL;
	bUP_TON_IN: BOOL;
	autocrosscut_error: TON;
	RS_TriggerReturn: RS;
	RS_TriggerCUT: RS;
	R_TRIG_0: R_TRIG;
	R_TRIG_1: R_TRIG;
	R_TRIG_2: R_TRIG;
	R_TRIG_3: R_TRIG;
	R_TRIG_4: R_TRIG;
	R_TRIG_5: R_TRIG;
	RS_TriggerCUT2: RS;
	R_TRIG_10: R_TRIG;
	R_TRIG_11: R_TRIG;
	R_TRIG_12: R_TRIG;
	RS_TriggerReturn2: RS;
	R_TRIG_13: R_TRIG;
	R_TRIG_14: R_TRIG;
	R_TRIG_15: R_TRIG;

	rCutSpeed: REAL;
	rReturnSpeed: REAL;
	rVFDMaxSpeed: REAL;
	rBufferSpeed: REAL;
	rSawOFFSpeed: REAL;
	rSpeedScaled: REAL;
	// speed test
	iSpeedTest: INT;
	rSawCurrentTest: REAL;
	TON_step10: TON;
	TON_step20: TON;
	TON_step30: TON;
	TON_step40: TON;
	TON_step50: TON;
	TON_step60: TON;
	TON_DownDelay: TON;
END_VAR

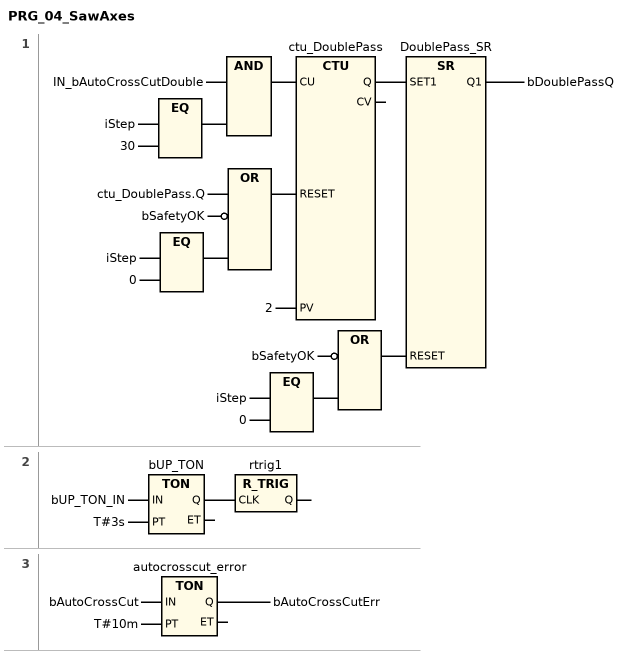
// NETWORK 1
ctu_DoublePass(
    CU := IN_bAutoCrossCutDouble AND iStep = 30,
    RESET := ctu_DoublePass.Q OR NOT bSafetyOK OR iStep = 0,
    PV := 2); // CTU
DoublePass_SR(SET1 := ctu_DoublePass.Q, RESET := NOT bSafetyOK OR iStep = 0); // SR
bDoublePassQ := DoublePass_SR.Q1;

// NETWORK 2
bUP_TON(IN := bUP_TON_IN, PT := T#3s); // TON
rtrig1(CLK := bUP_TON.Q); // R_TRIG

// NETWORK 3
autocrosscut_error(IN := bAutoCrossCut, PT := T#10m); // TON
bAutoCrossCutErr := autocrosscut_error.Q;

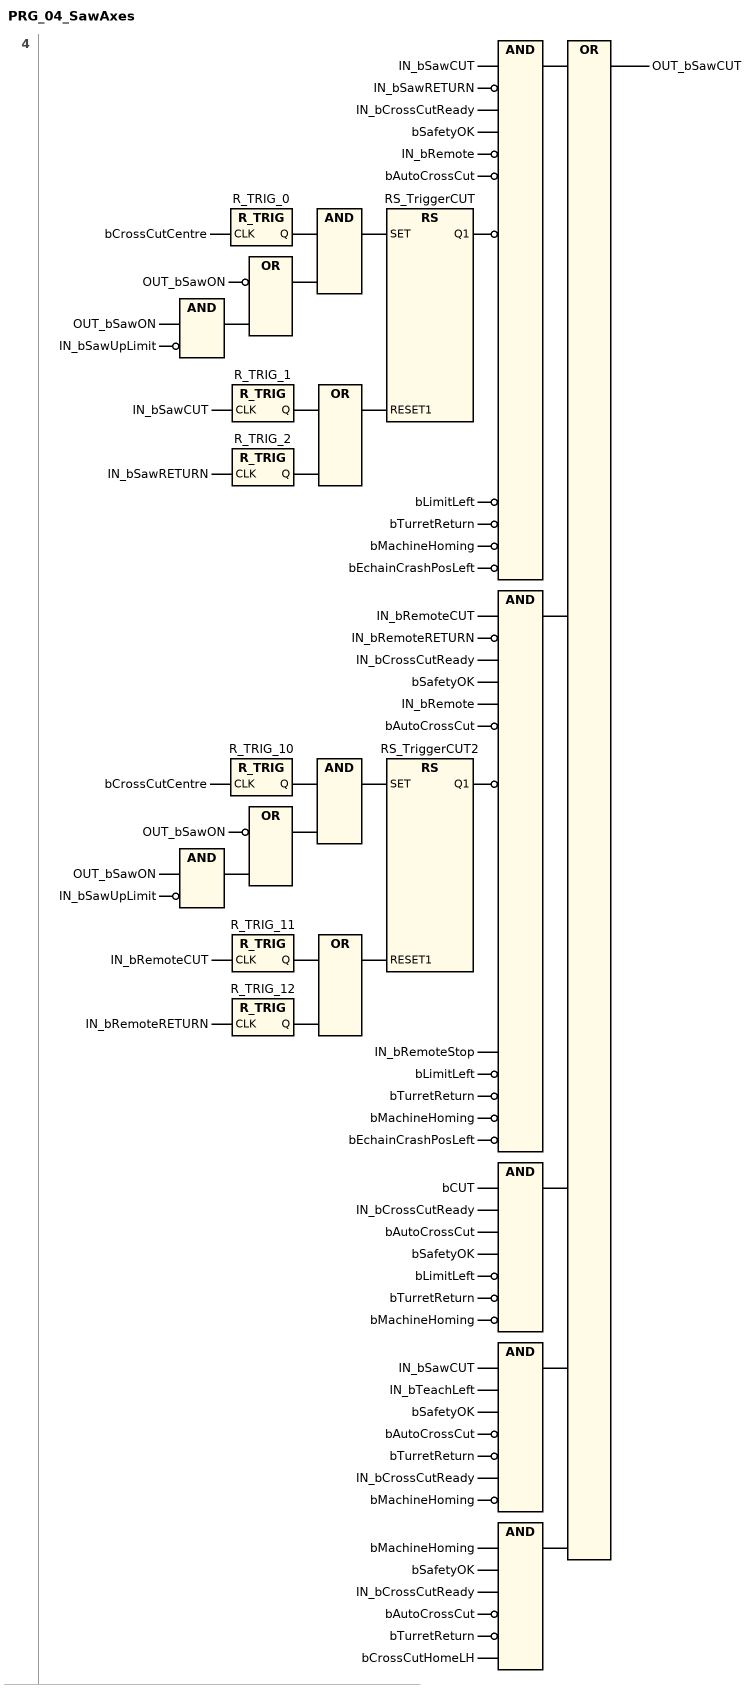
// NETWORK 4
R_TRIG_0(CLK := bCrossCutCentre); // R_TRIG
R_TRIG_1(CLK := IN_bSawCUT); // R_TRIG
R_TRIG_2(CLK := IN_bSawRETURN); // R_TRIG
RS_TriggerCUT(SET := R_TRIG_0.Q AND (NOT OUT_bSawON OR OUT_bSawON AND NOT IN_bSawUpLimit), RESET1 := R_TRIG_1.Q OR R_TRIG_2.Q); // RS
R_TRIG_10(CLK := bCrossCutCentre); // R_TRIG
R_TRIG_11(CLK := IN_bRemoteCUT); // R_TRIG
R_TRIG_12(CLK := IN_bRemoteRETURN); // R_TRIG
RS_TriggerCUT2(SET := R_TRIG_10.Q AND (NOT OUT_bSawON OR OUT_bSawON AND NOT IN_bSawUpLimit), RESET1 := R_TRIG_11.Q OR R_TRIG_12.Q); // RS
OUT_bSawCUT := IN_bSawCUT AND NOT IN_bSawRETURN AND IN_bCrossCutReady AND bSafetyOK AND NOT IN_bRemote AND NOT bAutoCrossCut AND NOT RS_TriggerCUT.Q1 AND NOT bLimitLeft AND NOT bTurretReturn AND NOT bMachineHoming AND NOT bEchainCrashPosLeft OR IN_bRemoteCUT AND NOT IN_bRemoteRETURN AND IN_bCrossCutReady AND bSafetyOK AND IN_bRemote AND NOT bAutoCrossCut AND NOT RS_TriggerCUT2.Q1 AND IN_bRemoteStop AND NOT bLimitLeft AND NOT bTurretReturn AND NOT bMachineHoming AND NOT bEchainCrashPosLeft OR bCUT AND IN_bCrossCutReady AND bAutoCrossCut AND bSafetyOK AND NOT bLimitLeft AND NOT bTurretReturn AND NOT bMachineHoming OR IN_bSawCUT AND IN_bTeachLeft AND bSafetyOK AND NOT bAutoCrossCut AND NOT bTurretReturn AND IN_bCrossCutReady AND NOT bMachineHoming OR bMachineHoming AND bSafetyOK AND IN_bCrossCutReady AND NOT bAutoCrossCut AND NOT bTurretReturn AND bCrossCutHomeLH;

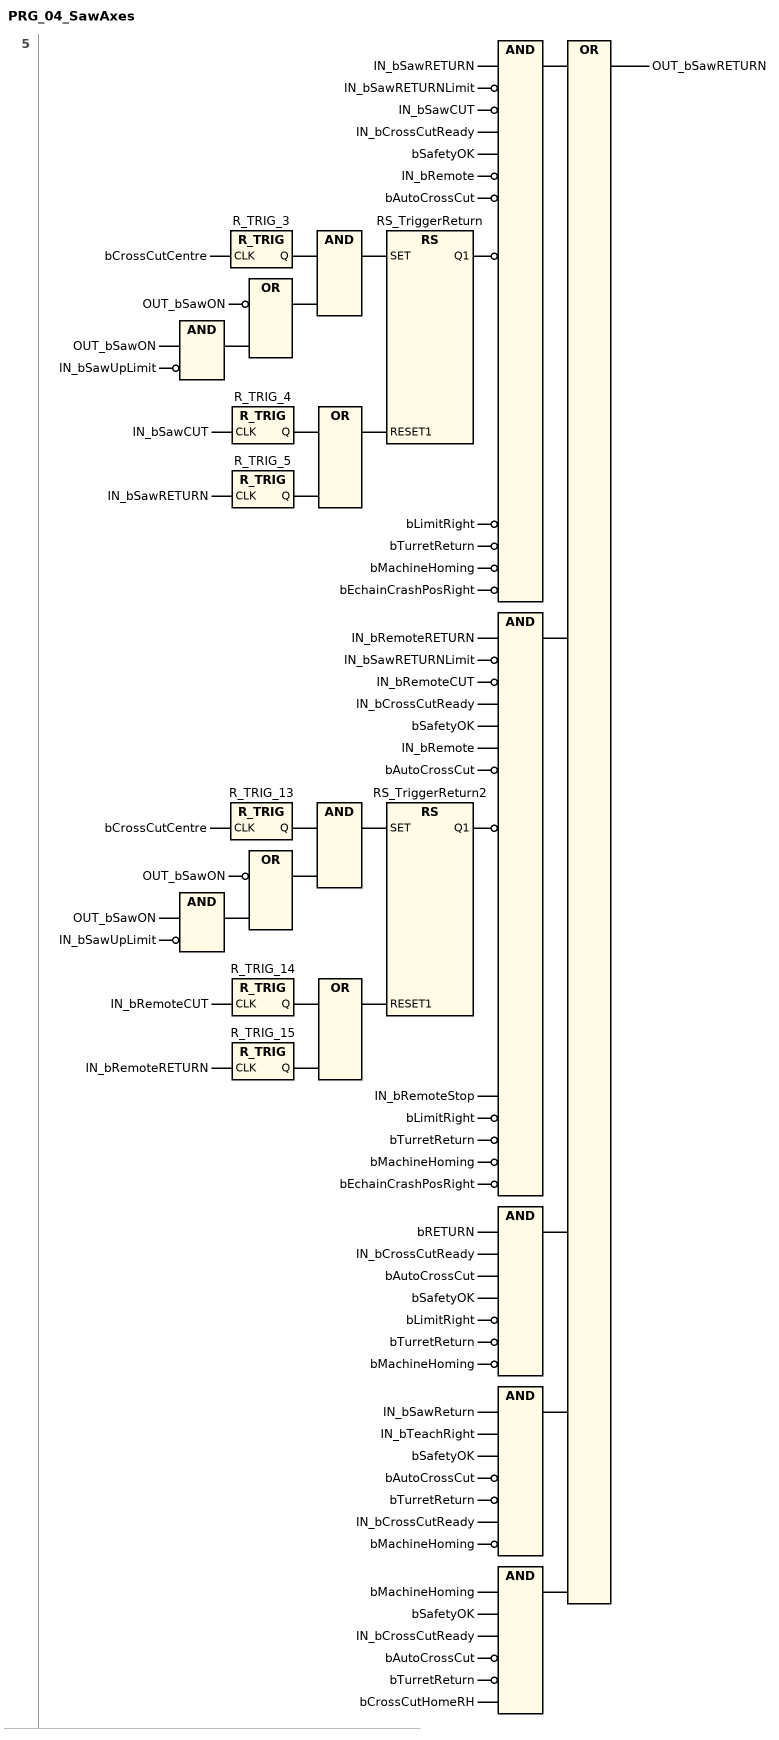
// NETWORK 5
R_TRIG_3(CLK := bCrossCutCentre); // R_TRIG
R_TRIG_4(CLK := IN_bSawCUT); // R_TRIG
R_TRIG_5(CLK := IN_bSawRETURN); // R_TRIG
RS_TriggerReturn(SET := R_TRIG_3.Q AND (NOT OUT_bSawON OR OUT_bSawON AND NOT IN_bSawUpLimit), RESET1 := R_TRIG_4.Q OR R_TRIG_5.Q); // RS
R_TRIG_13(CLK := bCrossCutCentre); // R_TRIG
R_TRIG_14(CLK := IN_bRemoteCUT); // R_TRIG
R_TRIG_15(CLK := IN_bRemoteRETURN); // R_TRIG
RS_TriggerReturn2(SET := R_TRIG_13.Q AND (NOT OUT_bSawON OR OUT_bSawON AND NOT IN_bSawUpLimit), RESET1 := R_TRIG_14.Q OR R_TRIG_15.Q); // RS
OUT_bSawRETURN := IN_bSawRETURN AND NOT IN_bSawRETURNLimit AND NOT IN_bSawCUT AND IN_bCrossCutReady AND bSafetyOK AND NOT IN_bRemote AND NOT bAutoCrossCut AND NOT RS_TriggerReturn.Q1 AND NOT bLimitRight AND NOT bTurretReturn AND NOT bMachineHoming AND NOT bEchainCrashPosRight OR IN_bRemoteRETURN AND NOT IN_bSawRETURNLimit AND NOT IN_bRemoteCUT AND IN_bCrossCutReady AND bSafetyOK AND IN_bRemote AND NOT bAutoCrossCut AND NOT RS_TriggerReturn2.Q1 AND IN_bRemoteStop AND NOT bLimitRight AND NOT bTurretReturn AND NOT bMachineHoming AND NOT bEchainCrashPosRight OR bRETURN AND IN_bCrossCutReady AND bAutoCrossCut AND bSafetyOK AND NOT bLimitRight AND NOT bTurretReturn AND NOT bMachineHoming OR IN_bSawReturn AND IN_bTeachRight AND bSafetyOK AND NOT bAutoCrossCut AND NOT bTurretReturn AND IN_bCrossCutReady AND NOT bMachineHoming OR bMachineHoming AND bSafetyOK AND IN_bCrossCutReady AND NOT bAutoCrossCut AND NOT bTurretReturn AND bCrossCutHomeRH;

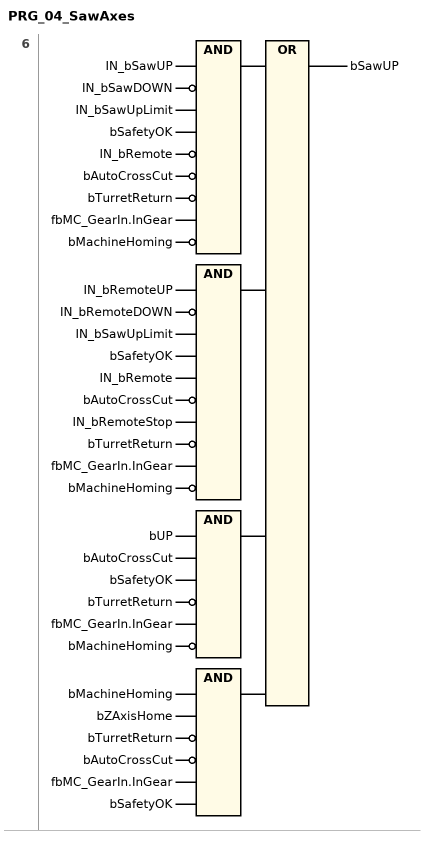
// NETWORK 6
bSawUP := IN_bSawUP AND NOT IN_bSawDOWN AND IN_bSawUpLimit AND bSafetyOK AND NOT IN_bRemote AND NOT bAutoCrossCut AND NOT bTurretReturn AND fbMC_GearIn.InGear AND NOT bMachineHoming OR IN_bRemoteUP AND NOT IN_bRemoteDOWN AND IN_bSawUpLimit AND bSafetyOK AND IN_bRemote AND NOT bAutoCrossCut AND IN_bRemoteStop AND NOT bTurretReturn AND fbMC_GearIn.InGear AND NOT bMachineHoming OR bUP AND bAutoCrossCut AND bSafetyOK AND NOT bTurretReturn AND fbMC_GearIn.InGear AND NOT bMachineHoming OR bMachineHoming AND bZAxisHome AND NOT bTurretReturn AND NOT bAutoCrossCut AND fbMC_GearIn.InGear AND bSafetyOK;

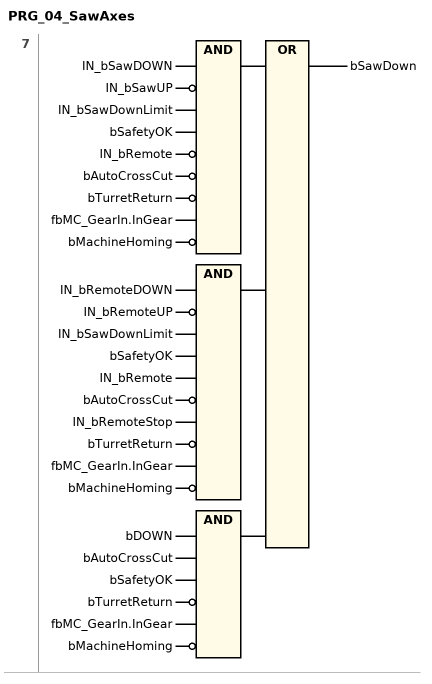
// NETWORK 7
bSawDown := IN_bSawDOWN AND NOT IN_bSawUP AND IN_bSawDownLimit AND bSafetyOK AND NOT IN_bRemote AND NOT bAutoCrossCut AND NOT bTurretReturn AND fbMC_GearIn.InGear AND NOT bMachineHoming OR IN_bRemoteDOWN AND NOT IN_bRemoteUP AND IN_bSawDownLimit AND bSafetyOK AND IN_bRemote AND NOT bAutoCrossCut AND IN_bRemoteStop AND NOT bTurretReturn AND fbMC_GearIn.InGear AND NOT bMachineHoming OR bDOWN AND bAutoCrossCut AND bSafetyOK AND NOT bTurretReturn AND fbMC_GearIn.InGear AND NOT bMachineHoming;

ACTION ACT_04_1_AutoCrossCut:
	IF		NOT bSafetyOK OR IN_FaultReset OR NOT OUT_bSawON
	THEN	iStep	:=	0;
	END_IF

	TON_DownDelay(IN:= , PT:= T#3S, Q=> , ET=> );
	IF		iStep <> 30 THEN
			TON_DownDelay.IN	:= FALSE ;
	END_IF
(* Double Pass counter BOOL *)
	IF		ctu_DoublePass.CV	=	1
	THEN	bDoublePassCountUp		:=	TRUE;
	ELSE	bDoublePassCountUp		:=	FALSE;
	END_IF

CASE iStep OF 
	0:		//	Step 0	:	Init step
				bAutoCrossCut	:= FALSE ;
				bUP				:= FALSE ;
				bDOWN			:= FALSE ;
				bCUT			:= FALSE ;
				bRETURN			:= FALSE ;
				bUP_TON_IN		:= FALSE ;
				
		IF
				bSafetyOK
				AND bTurret045Range
				AND OUT_bSawON
				AND (IN_bCrossCutLeft AND IN_bCrossCutRight AND NOT IN_bRemote)
				AND NOT (bTurretReturn OR bMachineHoming)
				AND NOT IN_bCarriageReference
		THEN
				bAutoCrossCut := TRUE	;
				iStep	:=		20		;
		ELSE
				bAutoCrossCut := FALSE	;
				iStep	:=		0		;
		END_IF

	20:		// Step 20	:	Saw RETURN movement
		IF 
				bAutoCrossCut
				AND bSafetyOK
				AND NOT bLimitRight
			
		THEN	bRETURN		:=	TRUE	;
		
		ELSE
				bRETURN		:=	FALSE	;
				iStep		:=	30		;
		END_IF
	
		IF 		NOT bSafetyOK
		THEN 	
				bRETURN		:=	FALSE	;
				iStep		:=	0		;
		END_IF
		
	30:		// Step 30	:	Saw DOWN movement
	ctu_DoublePass.CV;
		IF
				bAutoCrossCut
				AND bSafetyOK
				AND ((IN_bAutoCrossCutDouble AND IN_bDoublePassReference AND bDoublePassCountUp) 
					OR ( IN_bSawDownLimit AND (bDoublePassQ OR NOT bDoublePassCountUp)))
		THEN	
				bDOWN		:=	TRUE	;
		ELSE
				bDOWN		:=	FALSE	;
				TON_DownDelay.IN := TRUE ;
					IF TON_DownDelay.Q THEN
						iStep	:=	40		;
					END_IF
		END_IF
		
		IF 		NOT bSafetyOK
		THEN 	
				bDOWN		:=	FALSE	;
				iStep		:=	0		;
		END_IF
	
	40:		// Step 40	:	Saw CUT movement
		IF
				bAutoCrossCut
				AND bSafetyOK
				AND	NOT bLimitLeft
			THEN
				bCUT		:=	TRUE	;
		ELSE
				bCUT		:=	FALSE	;
				iStep		:=	50		;
		END_IF
		
		IF 		NOT bSafetyOK
			THEN 	
				bCUT		:=	FALSE	;
				iStep		:=	0		;
		END_IF
	
	50:		// Step 50	:	Saw UP movement		(* for double pass: only lift slightly, RETURN, then plunge all the way down *)
	ctu_DoublePass.CV;	
		IF
				IN_bAutoCrossCutDouble AND bDoublePassCountUp AND NOT bDoublePassQ
			THEN
				bUP_TON_IN	:=	TRUE	;
				bUP			:=	NOT bUP_TON.Q	;
				
				IF
					rtrig1.Q THEN
					iStep	:=	60	;
				END_IF
				
		ELSIF
				bAutoCrossCut
				AND bSafetyOK
				AND IN_bSawUpLimit
				AND ((bDoublePassQ AND NOT bDoublePassCountUp AND IN_bAutoCrossCutDouble) OR (NOT IN_bAutoCrossCutDouble))
			THEN
				bUP			:=	TRUE	;
		ELSE
				bUP			:=	FALSE	;
				iStep		:=	60		;
		END_IF
		
		IF 		NOT bSafetyOK
		THEN 	
				bUP			:=	FALSE	;
				iStep		:=	0		;
		END_IF
	
	60:		// Step 60	:	Saw RETURN movement (loop back to step 20 if double pass)
		IF
				IN_bAutoCrossCutDouble
				AND bDoublePassCountUp
		THEN
				iStep		:=	20		;
		ELSIF	
				bAutoCrossCut
				AND bSafetyOK
				AND NOT bCrossCutCentre
		THEN
				bRETURN		:=	TRUE	;
		ELSE
				bRETURN		:=	FALSE	;
				iStep		:=	0		;
		END_IF
	
END_CASE
END_ACTION

ACTION ACT_04_2_CrossCutSpeed:
// Cut and Return speed in VFD Hz
rCutSpeed := 5 ;
rReturnSpeed := 8.5 ;		
rVFDMaxSpeed := 20 ;		// set VFD P1-01 to this same Hz setting
rBufferSpeed := 2 ;
rSawOFFSpeed := 15 ;
rSpeedScaled := (INT_TO_REAL(OUT_iCrossCutFeedback) / 32767) * rVFDMaxSpeed ;
			
		IF fbSawCurrent.Out.rScaled < 40 THEN		// current feedback threshold
			rCrossCutSpeedMultiplier := 1 ;
		ELSIF fbSawCurrent.Out.rScaled > 40 AND fbSawCurrent.Out.rScaled < 55 THEN
			rCrossCutSpeedMultiplier := 0.75 ;
		ELSIF fbSawCurrent.Out.rScaled > 55 AND fbSawCurrent.Out.rScaled < 70 THEN
			rCrossCutSpeedMultiplier := 0.5 ;
		ELSIF fbSawCurrent.Out.rScaled > 70 AND fbSawCurrent.Out.rScaled < 85 THEN
			rCrossCutSpeedMultiplier := 0.4 ;
		ELSIF fbSawCurrent.Out.rScaled > 85 THEN
			rCrossCutSpeedMultiplier := 0.2 ;
		END_IF

IF OUT_bSawRETURN AND NOT OUT_bSawCUT AND NOT bApproachingLimitRight AND OUT_bSawON THEN	// Return speed if Saw blade is ON
	OUT_iCrossCutFeedback := REAL_TO_INT((rReturnSpeed / rVFDMaxSpeed) * 32767) ;
																	
ELSIF OUT_bSawCUT AND NOT OUT_bSawRETURN AND NOT bApproachingLimitLeft AND OUT_bSawON THEN	// Cut speed if Saw blade is ON
	OUT_iCrossCutFeedback := REAL_TO_INT(((rCutSpeed * rCrossCutSpeedMultiplier) / rVFDMaxSpeed) * 32767) ; // ##### CURRENT FEEDBACK #####
	
ELSIF ((OUT_bSawCUT AND bApproachingLimitLeft) OR (OUT_bSawRETURN AND bApproachingLimitRight))  THEN	// Buffer speed as the blade approaches the edge limits
	OUT_iCrossCutFeedback := REAL_TO_INT((rBufferSpeed / rVFDMaxSpeed) * 32767) ;
	
ELSIF ((OUT_bSawCUT AND NOT bApproachingLimitLeft) OR (OUT_bSawRETURN AND NOT bApproachingLimitRight)) AND NOT OUT_bSawON THEN // Cut and Return speed if Saw blade OFF
	OUT_iCrossCutFeedback := REAL_TO_INT((rSawOFFSpeed / rVFDMaxSpeed) * 32767) ;
ELSE
	OUT_iCrossCutFeedback := 0 ;
END_IF

(*		// Current Feedback Test
IF NOT bSafetyOK THEN
	iSpeedTest := 0;
END_IF

CASE iSpeedTest OF
	0: // 0 A before startup
		rSawCurrentTest := 0;
		TON_step10	.IN	:= FALSE ;
		TON_step20	.IN	:= FALSE ;
		TON_step30	.IN	:= FALSE ;
		TON_step40	.IN	:= FALSE ;
		TON_step50	.IN	:= FALSE ;
		TON_step60	.IN	:= FALSE ;
	10: // constant 33 A after startup for 3 sec
		TON_step10(IN:= , PT:= T#3S, Q=> , ET=> );
		TON_step10.IN := TRUE;
		rSawCurrentTest := 33;
		IF TON_step10.Q THEN
			iSpeedTest := 20;
		END_IF
	20: // increase to 38 A for 3 sec
		TON_step20(IN:= , PT:= T#3S, Q=> , ET=> );
		TON_step20.IN := TRUE;
		rSawCurrentTest := 38;
		IF TON_step20.Q THEN
			iSpeedTest := 30;
		END_IF
	30: // increase to 45 A for 2 sec
		TON_step30(IN:= , PT:= T#2S, Q=> , ET=> );
		TON_step30.IN := TRUE;
		rSawCurrentTest := 45;
		IF TON_step30.Q THEN
			iSpeedTest := 40;
		END_IF
	40: // decrease back to 38 A for 2 sec
		TON_step40(IN:= , PT:= T#2S, Q=> , ET=> );
		TON_step40.IN := TRUE;
		rSawCurrentTest := 38;
		IF TON_step40.Q THEN
			iSpeedTest := 50;
		END_IF
	50: // spike to 55 A for 0.5 sec
		TON_step50(IN:= , PT:= T#2S, Q=> , ET=> );
		TON_step50.IN := TRUE;
		rSawCurrentTest := 55;
		IF TON_step50.Q THEN
			iSpeedTest := 60;
		END_IF
	60: // decrease back to 38 A to finish the cut
		TON_step60(IN:= , PT:= T#2S, Q=> , ET=> );
		TON_step60.IN := TRUE;
		rSawCurrentTest := 38;
		IF TON_step60.Q THEN
			iSpeedTest := 0;
		END_IF
	
END_CASE
*)
END_ACTION

END_PROGRAM

// ---- POUs/MAIN FUNCTIONS/PRG_05_Turret_Carriage.TcPOU
PROGRAM PRG_05_Turret_Carriage
VAR
	R_TRIG_0: R_TRIG;
	R_TRIG_1: R_TRIG;
	F_TRIG_2: F_TRIG;
	F_TRIG_4: F_TRIG;
	RS_TriggerStopCCW: RS;
	R_TRIG_12: R_TRIG;
	RS_TriggerStopCW: RS;
	R_TRIG_15: R_TRIG;
	R_TRIG_18: R_TRIG;
	R_TRIG_19: R_TRIG;
	R_TRIG_20: R_TRIG;
	R_TRIG_21: R_TRIG;
	R_TRIG_22: R_TRIG;
	TOF_SwitchDelay: TOF;
	R_TRIG_23: R_TRIG;
	R_TRIG_24: R_TRIG;
	R_TRIG_25: R_TRIG;
	R_TRIG_26: R_TRIG;
	F_TRIG_0: F_TRIG;
	F_TRIG_1: F_TRIG;
END_VAR
VAR // added by the converter: edge detectors and wires of the graphical bodies
    _w1, _w2 : BOOL;
END_VAR

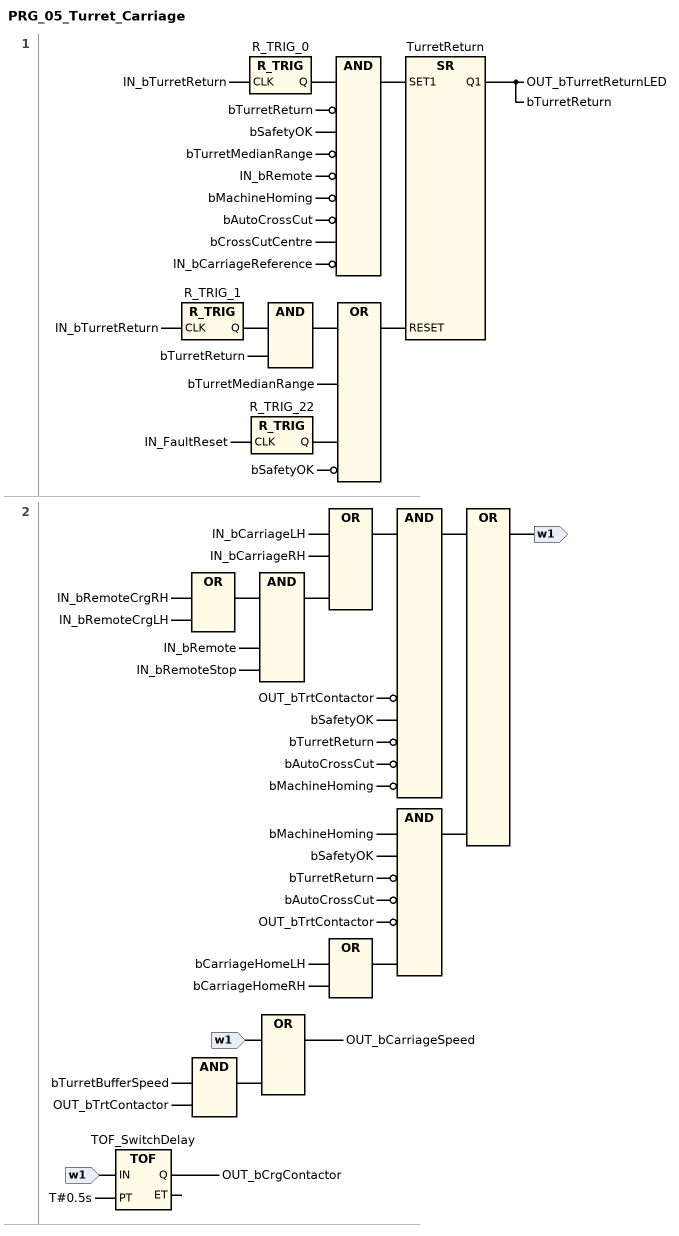
// NETWORK 1
R_TRIG_0(CLK := IN_bTurretReturn); // R_TRIG
R_TRIG_1(CLK := IN_bTurretReturn); // R_TRIG
R_TRIG_22(CLK := IN_FaultReset); // R_TRIG
TurretReturn(SET1 := R_TRIG_0.Q AND NOT bTurretReturn AND bSafetyOK AND NOT bTurretMedianRange AND NOT IN_bRemote AND NOT bMachineHoming AND NOT bAutoCrossCut AND bCrossCutCentre AND NOT IN_bCarriageReference, RESET := R_TRIG_1.Q AND bTurretReturn OR bTurretMedianRange OR R_TRIG_22.Q OR NOT bSafetyOK); // SR
OUT_bTurretReturnLED := TurretReturn.Q1;
bTurretReturn := TurretReturn.Q1;

// NETWORK 2
_w1 := (IN_bCarriageLH OR IN_bCarriageRH OR (IN_bRemoteCrgRH OR IN_bRemoteCrgLH) AND IN_bRemote AND IN_bRemoteStop) AND NOT OUT_bTrtContactor AND bSafetyOK AND NOT bTurretReturn AND NOT bAutoCrossCut AND NOT bMachineHoming OR bMachineHoming AND bSafetyOK AND NOT bTurretReturn AND NOT bAutoCrossCut AND NOT OUT_bTrtContactor AND (bCarriageHomeLH OR bCarriageHomeRH);
OUT_bCarriageSpeed := _w1 OR bTurretBufferSpeed AND OUT_bTrtContactor;
TOF_SwitchDelay(IN := _w1, PT := T#0.5s); // TOF
OUT_bCrgContactor := TOF_SwitchDelay.Q;

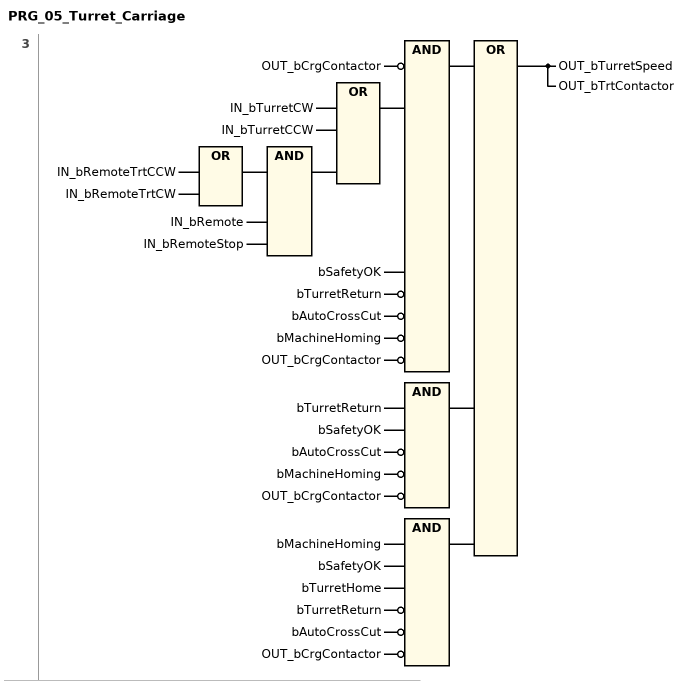
// NETWORK 3
_w2 := NOT OUT_bCrgContactor AND (IN_bTurretCW OR IN_bTurretCCW OR (IN_bRemoteTrtCCW OR IN_bRemoteTrtCW) AND IN_bRemote AND IN_bRemoteStop) AND bSafetyOK AND NOT bTurretReturn AND NOT bAutoCrossCut AND NOT bMachineHoming AND NOT OUT_bCrgContactor OR bTurretReturn AND bSafetyOK AND NOT bAutoCrossCut AND NOT bMachineHoming AND NOT OUT_bCrgContactor OR bMachineHoming AND bSafetyOK AND bTurretHome AND NOT bTurretReturn AND NOT bAutoCrossCut AND NOT OUT_bCrgContactor;
OUT_bTurretSpeed := _w2;
OUT_bTrtContactor := _w2;

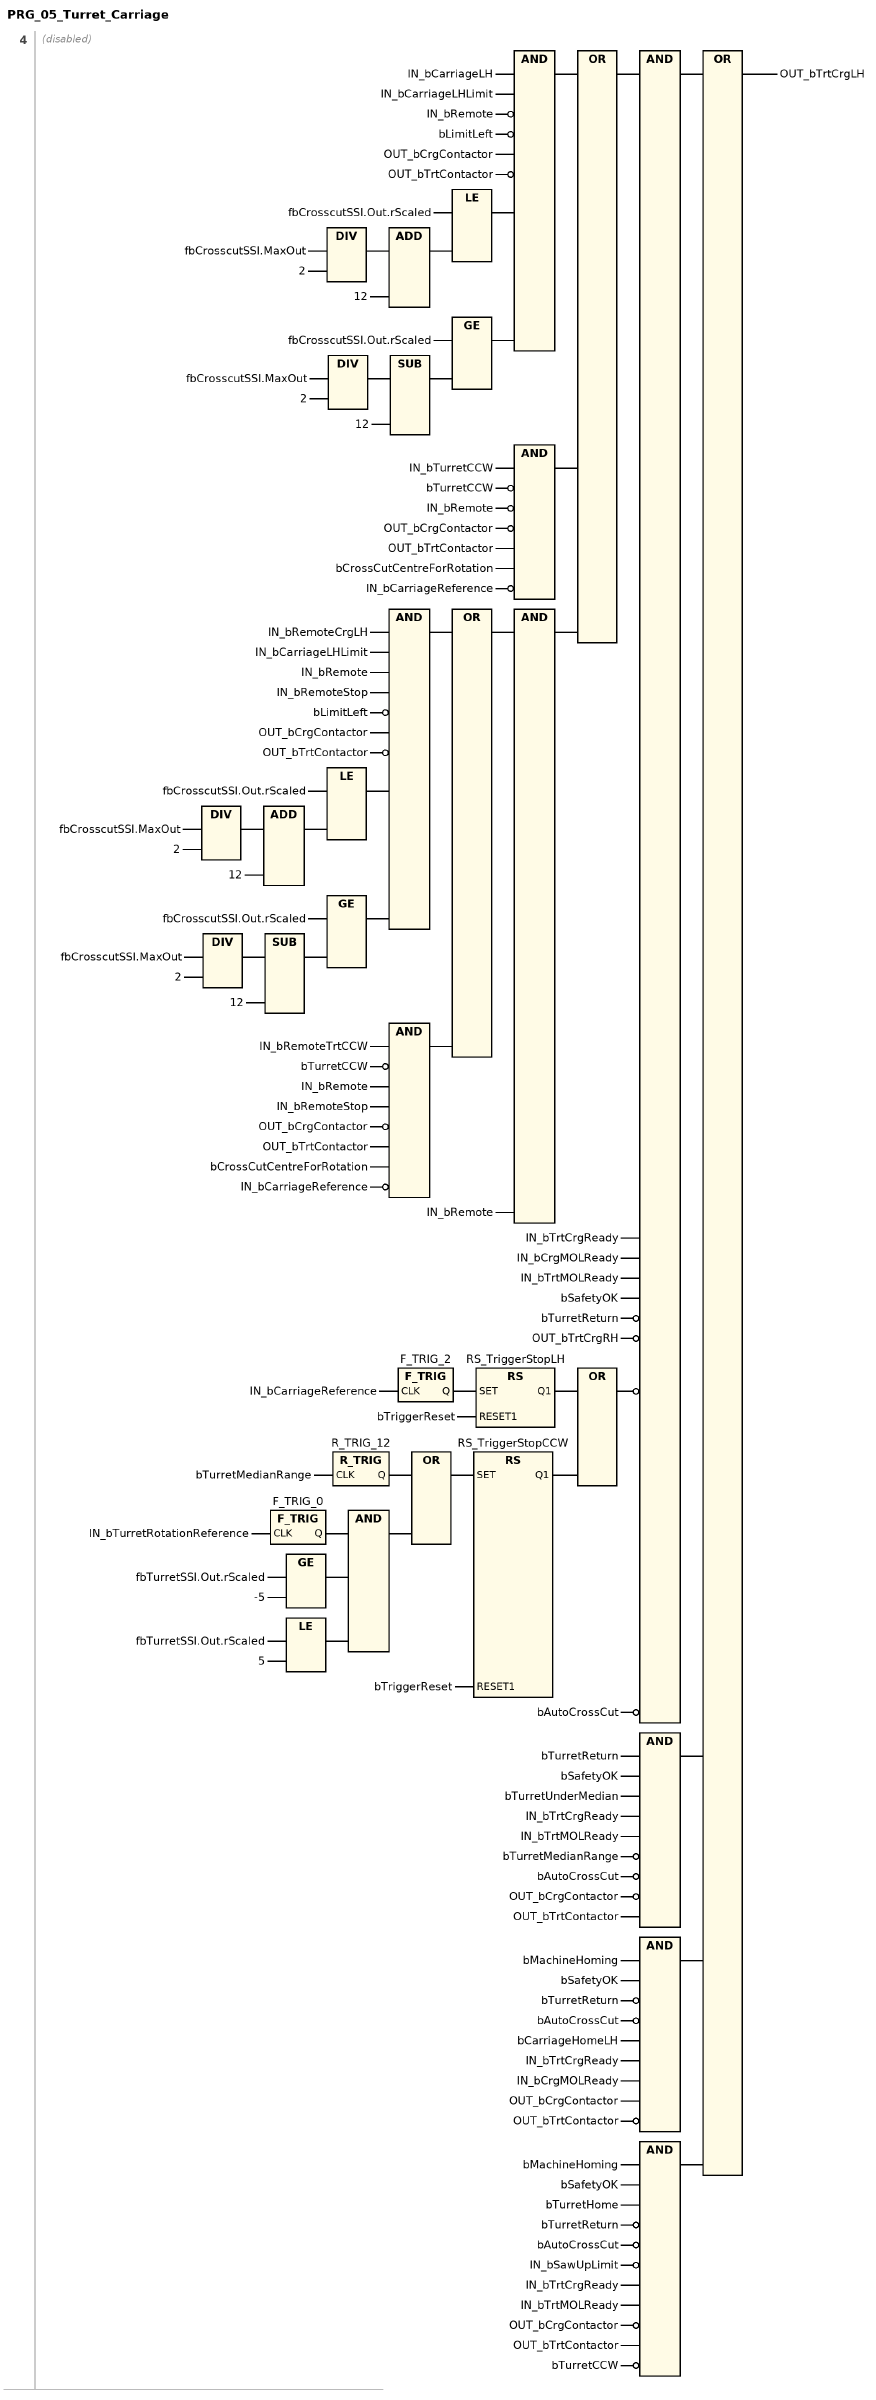
// NETWORK 4 (disabled)
// F_TRIG_2(CLK := IN_bCarriageReference); // F_TRIG
// RS_TriggerStopLH(SET := F_TRIG_2.Q, RESET1 := bTriggerReset); // RS
// R_TRIG_12(CLK := bTurretMedianRange); // R_TRIG
// F_TRIG_0(CLK := IN_bTurretRotationReference); // F_TRIG
// RS_TriggerStopCCW(SET := R_TRIG_12.Q OR F_TRIG_0.Q AND fbTurretSSI.Out.rScaled >= -5 AND fbTurretSSI.Out.rScaled <= 5, RESET1 := bTriggerReset); // RS
// OUT_bTrtCrgLH := (IN_bCarriageLH AND IN_bCarriageLHLimit AND NOT IN_bRemote AND NOT bLimitLeft AND OUT_bCrgContactor AND NOT OUT_bTrtContactor AND fbCrosscutSSI.Out.rScaled <= fbCrosscutSSI.MaxOut / 2 + 12 AND fbCrosscutSSI.Out.rScaled >= fbCrosscutSSI.MaxOut / 2 - 12 OR IN_bTurretCCW AND NOT bTurretCCW AND NOT IN_bRemote AND NOT OUT_bCrgContactor AND OUT_bTrtContactor AND bCrossCutCentreForRotation AND NOT IN_bCarriageReference OR (IN_bRemoteCrgLH AND IN_bCarriageLHLimit AND IN_bRemote AND IN_bRemoteStop AND NOT bLimitLeft AND OUT_bCrgContactor AND NOT OUT_bTrtContactor AND fbCrosscutSSI.Out.rScaled <= fbCrosscutSSI.MaxOut / 2 + 12 AND fbCrosscutSSI.Out.rScaled >= fbCrosscutSSI.MaxOut / 2 - 12 OR IN_bRemoteTrtCCW AND NOT bTurretCCW AND IN_bRemote AND IN_bRemoteStop AND NOT OUT_bCrgContactor AND OUT_bTrtContactor AND bCrossCutCentreForRotation AND NOT IN_bCarriageReference) AND IN_bRemote) AND IN_bTrtCrgReady AND IN_bCrgMOLReady AND IN_bTrtMOLReady AND bSafetyOK AND NOT bTurretReturn AND NOT OUT_bTrtCrgRH AND NOT (RS_TriggerStopLH.Q1 OR RS_TriggerStopCCW.Q1) AND NOT bAutoCrossCut OR bTurretReturn AND bSafetyOK AND bTurretUnderMedian AND IN_bTrtCrgReady AND IN_bTrtMOLReady AND NOT bTurretMedianRange AND NOT bAutoCrossCut AND NOT OUT_bCrgContactor AND OUT_bTrtContactor OR bMachineHoming AND bSafetyOK AND NOT bTurretReturn AND NOT bAutoCrossCut AND bCarriageHomeLH AND IN_bTrtCrgReady AND IN_bCrgMOLReady AND OUT_bCrgContactor AND NOT OUT_bTrtContactor OR bMachineHoming AND bSafetyOK AND bTurretHome AND NOT bTurretReturn AND NOT bAutoCrossCut AND NOT IN_bSawUpLimit AND IN_bTrtCrgReady AND IN_bTrtMOLReady AND NOT OUT_bCrgContactor AND OUT_bTrtContactor AND NOT bTurretCCW;

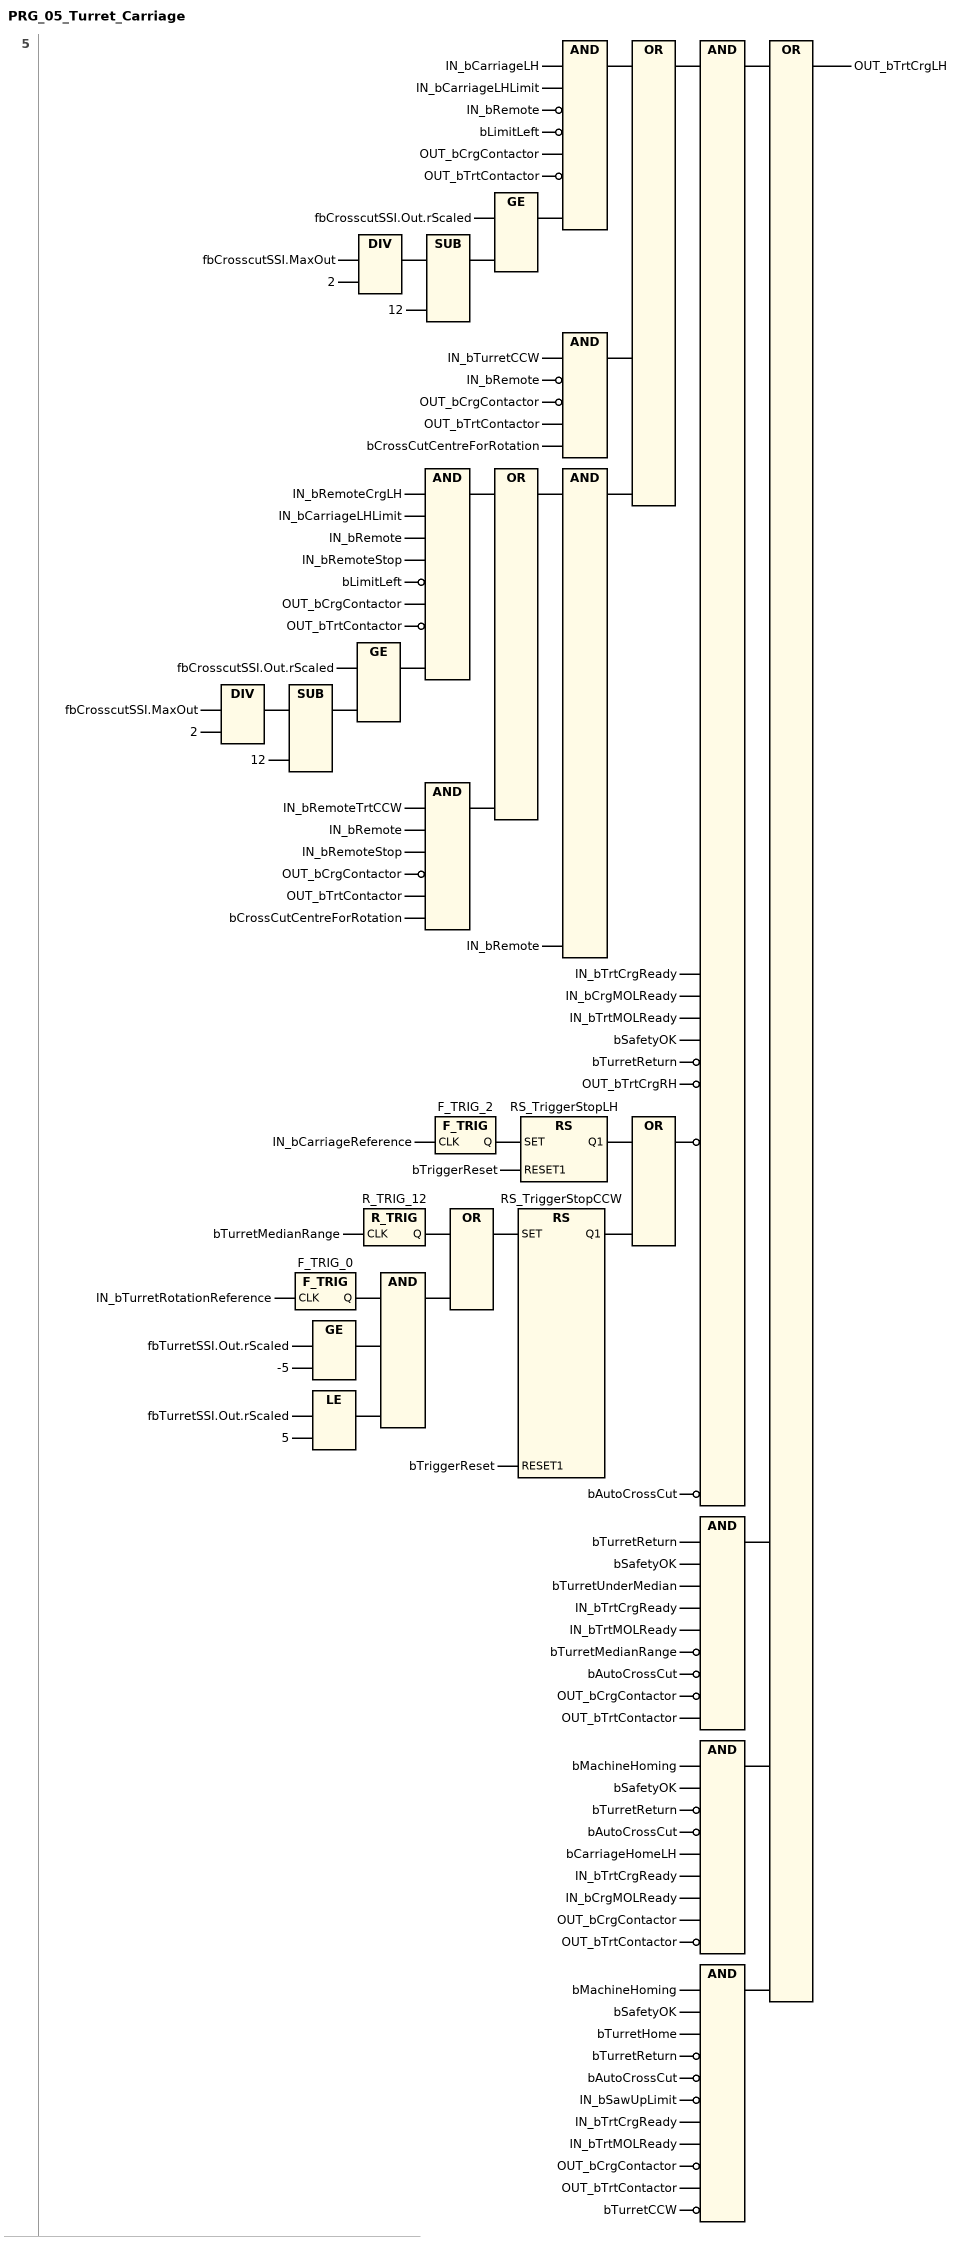
// NETWORK 5
F_TRIG_2(CLK := IN_bCarriageReference); // F_TRIG
RS_TriggerStopLH(SET := F_TRIG_2.Q, RESET1 := bTriggerReset); // RS
R_TRIG_12(CLK := bTurretMedianRange); // R_TRIG
F_TRIG_0(CLK := IN_bTurretRotationReference); // F_TRIG
RS_TriggerStopCCW(SET := R_TRIG_12.Q OR F_TRIG_0.Q AND fbTurretSSI.Out.rScaled >= -5 AND fbTurretSSI.Out.rScaled <= 5, RESET1 := bTriggerReset); // RS
OUT_bTrtCrgLH := (IN_bCarriageLH AND IN_bCarriageLHLimit AND NOT IN_bRemote AND NOT bLimitLeft AND OUT_bCrgContactor AND NOT OUT_bTrtContactor AND fbCrosscutSSI.Out.rScaled >= fbCrosscutSSI.MaxOut / 2 - 12 OR IN_bTurretCCW AND NOT IN_bRemote AND NOT OUT_bCrgContactor AND OUT_bTrtContactor AND bCrossCutCentreForRotation OR (IN_bRemoteCrgLH AND IN_bCarriageLHLimit AND IN_bRemote AND IN_bRemoteStop AND NOT bLimitLeft AND OUT_bCrgContactor AND NOT OUT_bTrtContactor AND fbCrosscutSSI.Out.rScaled >= fbCrosscutSSI.MaxOut / 2 - 12 OR IN_bRemoteTrtCCW AND IN_bRemote AND IN_bRemoteStop AND NOT OUT_bCrgContactor AND OUT_bTrtContactor AND bCrossCutCentreForRotation) AND IN_bRemote) AND IN_bTrtCrgReady AND IN_bCrgMOLReady AND IN_bTrtMOLReady AND bSafetyOK AND NOT bTurretReturn AND NOT OUT_bTrtCrgRH AND NOT (RS_TriggerStopLH.Q1 OR RS_TriggerStopCCW.Q1) AND NOT bAutoCrossCut OR bTurretReturn AND bSafetyOK AND bTurretUnderMedian AND IN_bTrtCrgReady AND IN_bTrtMOLReady AND NOT bTurretMedianRange AND NOT bAutoCrossCut AND NOT OUT_bCrgContactor AND OUT_bTrtContactor OR bMachineHoming AND bSafetyOK AND NOT bTurretReturn AND NOT bAutoCrossCut AND bCarriageHomeLH AND IN_bTrtCrgReady AND IN_bCrgMOLReady AND OUT_bCrgContactor AND NOT OUT_bTrtContactor OR bMachineHoming AND bSafetyOK AND bTurretHome AND NOT bTurretReturn AND NOT bAutoCrossCut AND NOT IN_bSawUpLimit AND IN_bTrtCrgReady AND IN_bTrtMOLReady AND NOT OUT_bCrgContactor AND OUT_bTrtContactor AND NOT bTurretCCW;

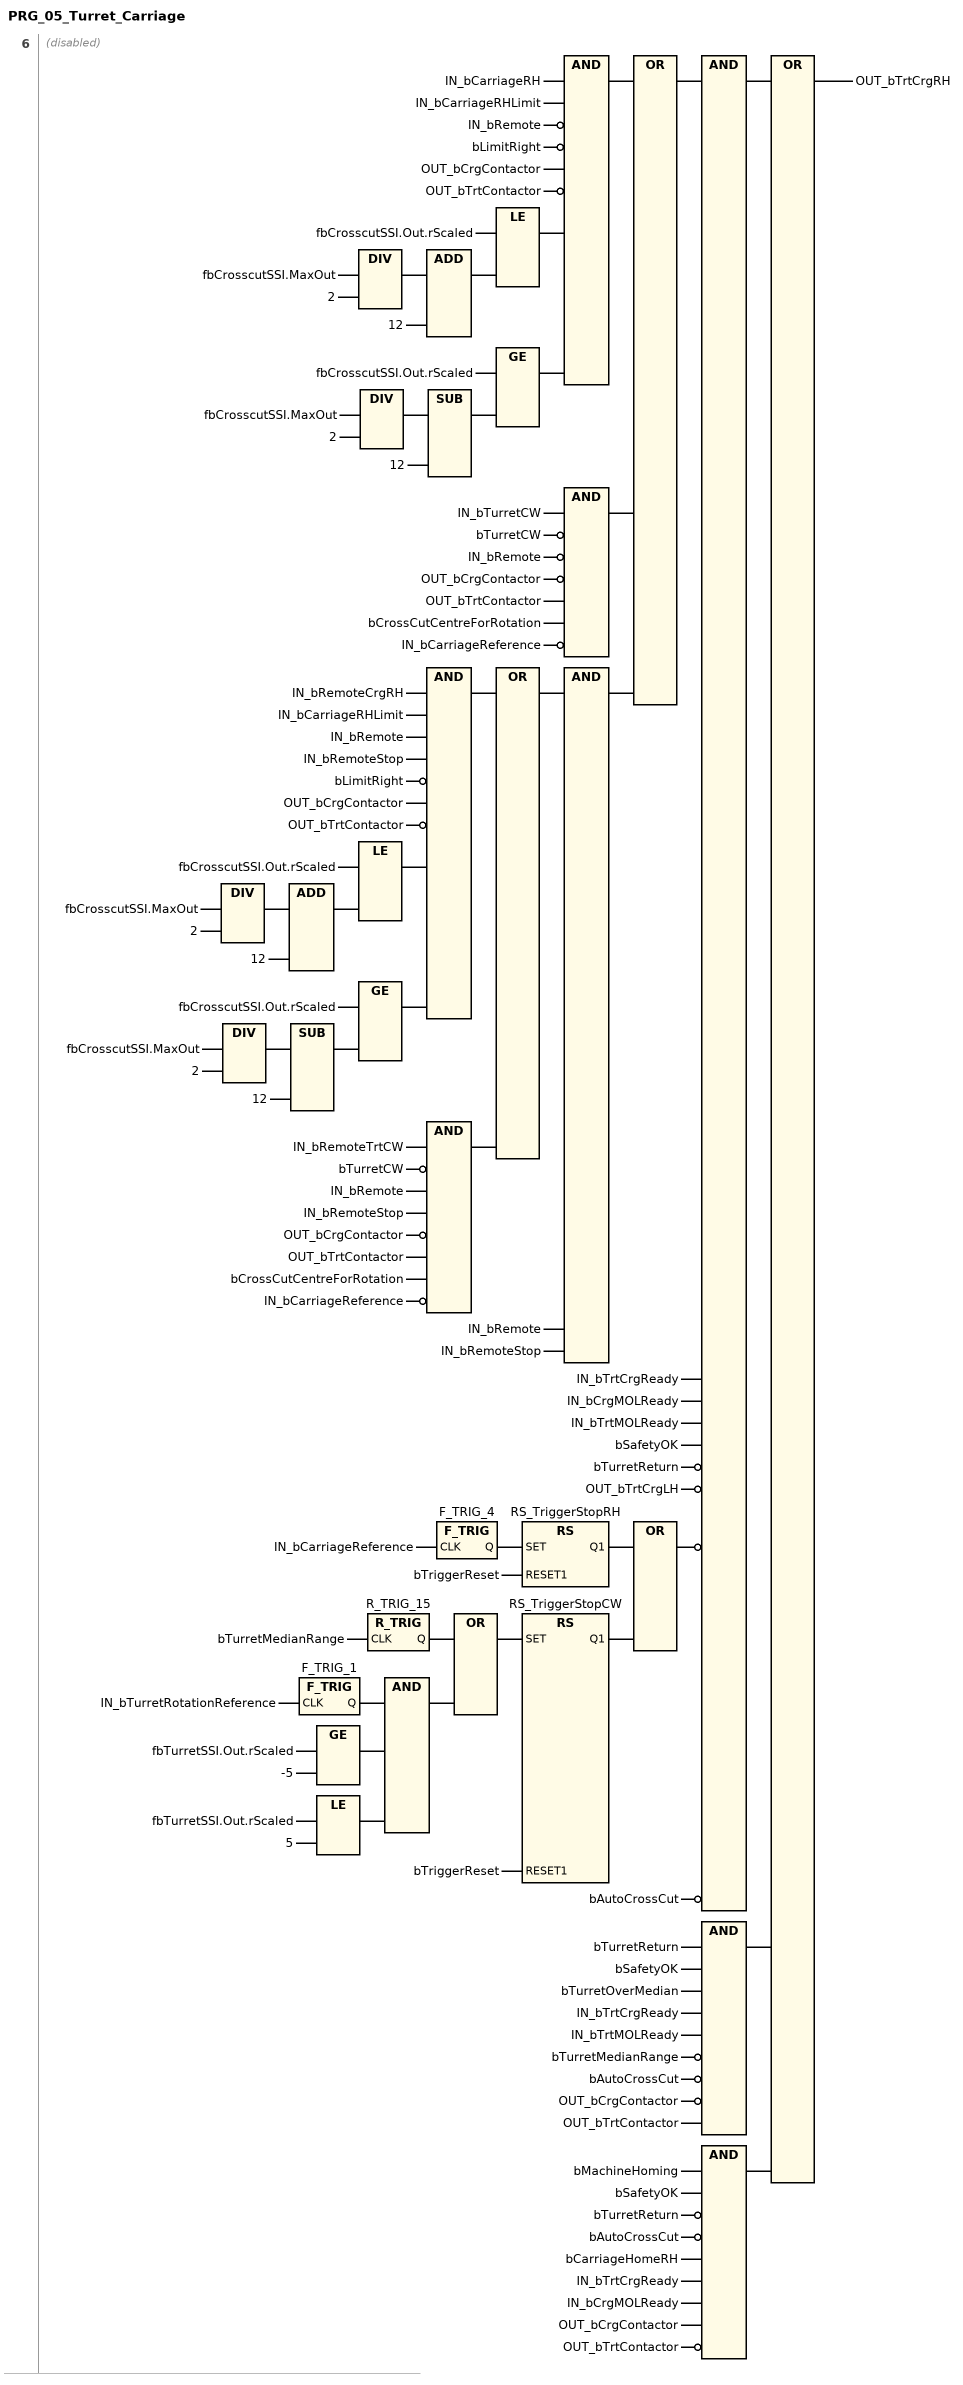
// NETWORK 6 (disabled)
// F_TRIG_4(CLK := IN_bCarriageReference); // F_TRIG
// RS_TriggerStopRH(SET := F_TRIG_4.Q, RESET1 := bTriggerReset); // RS
// R_TRIG_15(CLK := bTurretMedianRange); // R_TRIG
// F_TRIG_1(CLK := IN_bTurretRotationReference); // F_TRIG
// RS_TriggerStopCW(SET := R_TRIG_15.Q OR F_TRIG_1.Q AND fbTurretSSI.Out.rScaled >= -5 AND fbTurretSSI.Out.rScaled <= 5, RESET1 := bTriggerReset); // RS
// OUT_bTrtCrgRH := (IN_bCarriageRH AND IN_bCarriageRHLimit AND NOT IN_bRemote AND NOT bLimitRight AND OUT_bCrgContactor AND NOT OUT_bTrtContactor AND fbCrosscutSSI.Out.rScaled <= fbCrosscutSSI.MaxOut / 2 + 12 AND fbCrosscutSSI.Out.rScaled >= fbCrosscutSSI.MaxOut / 2 - 12 OR IN_bTurretCW AND NOT bTurretCW AND NOT IN_bRemote AND NOT OUT_bCrgContactor AND OUT_bTrtContactor AND bCrossCutCentreForRotation AND NOT IN_bCarriageReference OR (IN_bRemoteCrgRH AND IN_bCarriageRHLimit AND IN_bRemote AND IN_bRemoteStop AND NOT bLimitRight AND OUT_bCrgContactor AND NOT OUT_bTrtContactor AND fbCrosscutSSI.Out.rScaled <= fbCrosscutSSI.MaxOut / 2 + 12 AND fbCrosscutSSI.Out.rScaled >= fbCrosscutSSI.MaxOut / 2 - 12 OR IN_bRemoteTrtCW AND NOT bTurretCW AND IN_bRemote AND IN_bRemoteStop AND NOT OUT_bCrgContactor AND OUT_bTrtContactor AND bCrossCutCentreForRotation AND NOT IN_bCarriageReference) AND IN_bRemote AND IN_bRemoteStop) AND IN_bTrtCrgReady AND IN_bCrgMOLReady AND IN_bTrtMOLReady AND bSafetyOK AND NOT bTurretReturn AND NOT OUT_bTrtCrgLH AND NOT (RS_TriggerStopRH.Q1 OR RS_TriggerStopCW.Q1) AND NOT bAutoCrossCut OR bTurretReturn AND bSafetyOK AND bTurretOverMedian AND IN_bTrtCrgReady AND IN_bTrtMOLReady AND NOT bTurretMedianRange AND NOT bAutoCrossCut AND NOT OUT_bCrgContactor AND OUT_bTrtContactor OR bMachineHoming AND bSafetyOK AND NOT bTurretReturn AND NOT bAutoCrossCut AND bCarriageHomeRH AND IN_bTrtCrgReady AND IN_bCrgMOLReady AND OUT_bCrgContactor AND NOT OUT_bTrtContactor;

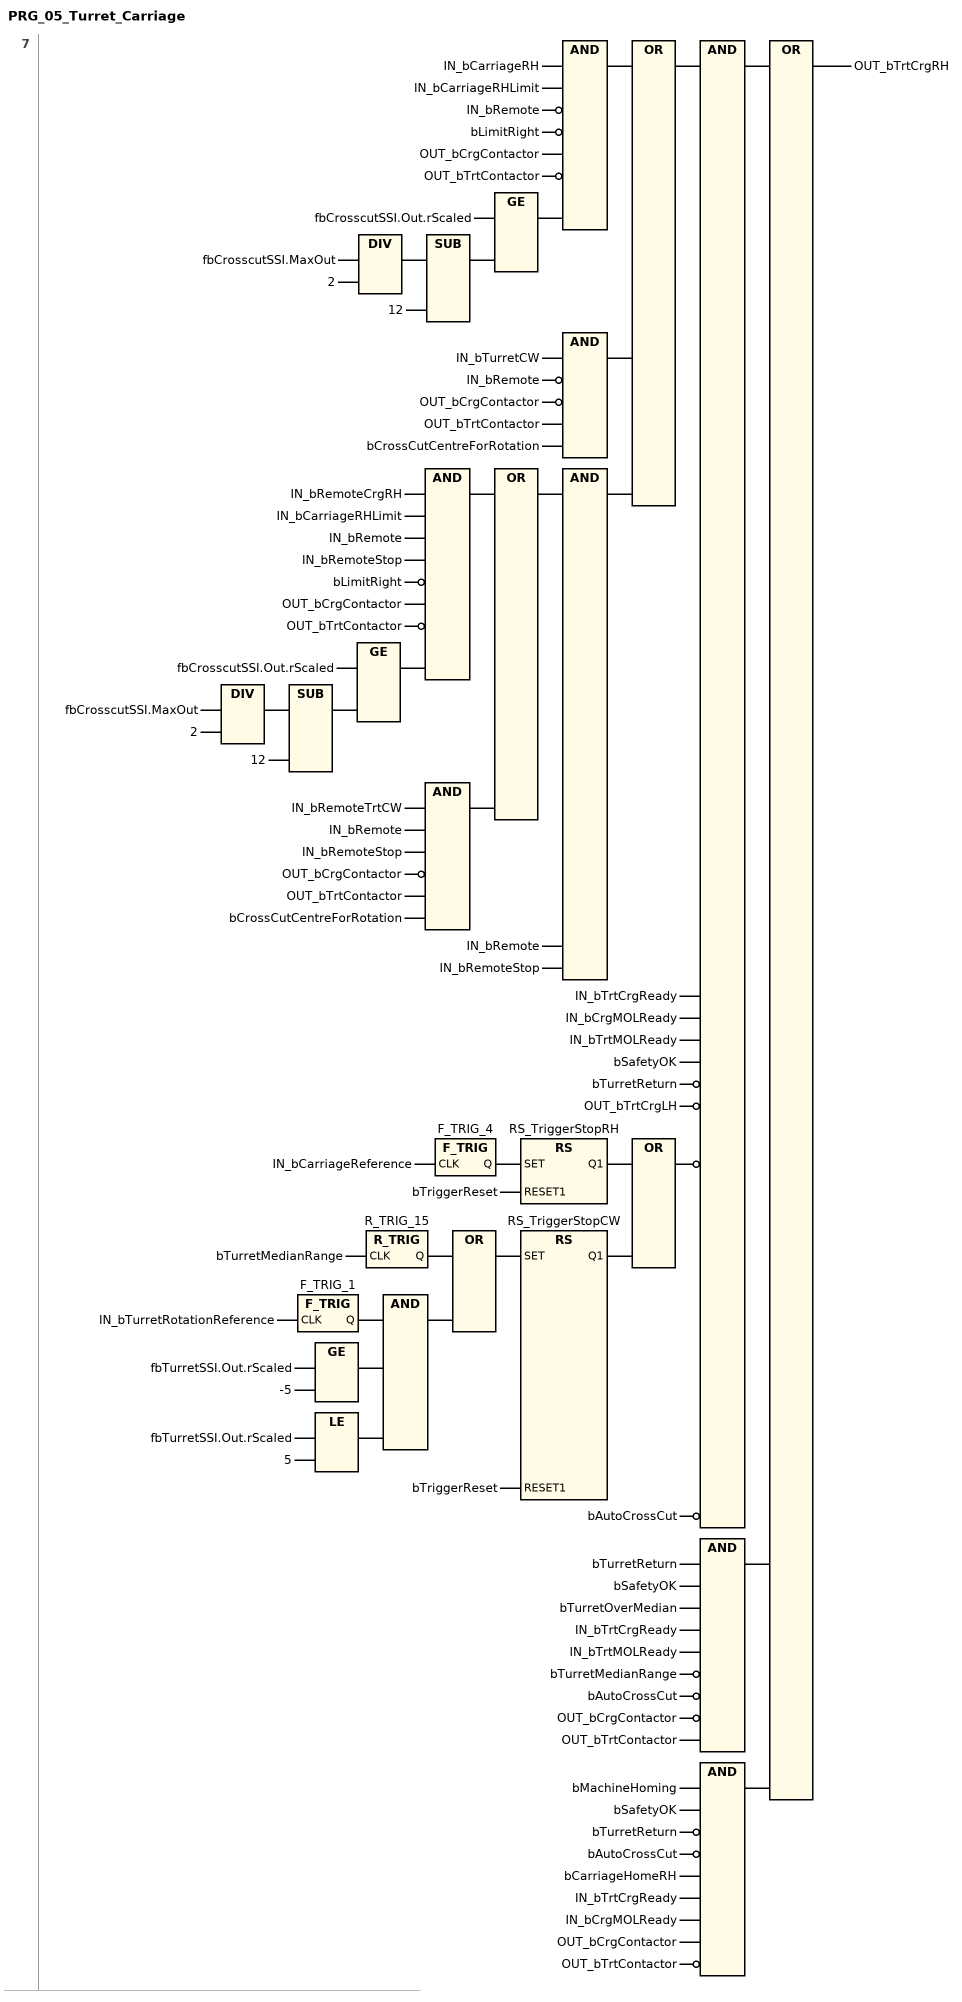
// NETWORK 7
F_TRIG_4(CLK := IN_bCarriageReference); // F_TRIG
RS_TriggerStopRH(SET := F_TRIG_4.Q, RESET1 := bTriggerReset); // RS
R_TRIG_15(CLK := bTurretMedianRange); // R_TRIG
F_TRIG_1(CLK := IN_bTurretRotationReference); // F_TRIG
RS_TriggerStopCW(SET := R_TRIG_15.Q OR F_TRIG_1.Q AND fbTurretSSI.Out.rScaled >= -5 AND fbTurretSSI.Out.rScaled <= 5, RESET1 := bTriggerReset); // RS
OUT_bTrtCrgRH := (IN_bCarriageRH AND IN_bCarriageRHLimit AND NOT IN_bRemote AND NOT bLimitRight AND OUT_bCrgContactor AND NOT OUT_bTrtContactor AND fbCrosscutSSI.Out.rScaled >= fbCrosscutSSI.MaxOut / 2 - 12 OR IN_bTurretCW AND NOT IN_bRemote AND NOT OUT_bCrgContactor AND OUT_bTrtContactor AND bCrossCutCentreForRotation OR (IN_bRemoteCrgRH AND IN_bCarriageRHLimit AND IN_bRemote AND IN_bRemoteStop AND NOT bLimitRight AND OUT_bCrgContactor AND NOT OUT_bTrtContactor AND fbCrosscutSSI.Out.rScaled >= fbCrosscutSSI.MaxOut / 2 - 12 OR IN_bRemoteTrtCW AND IN_bRemote AND IN_bRemoteStop AND NOT OUT_bCrgContactor AND OUT_bTrtContactor AND bCrossCutCentreForRotation) AND IN_bRemote AND IN_bRemoteStop) AND IN_bTrtCrgReady AND IN_bCrgMOLReady AND IN_bTrtMOLReady AND bSafetyOK AND NOT bTurretReturn AND NOT OUT_bTrtCrgLH AND NOT (RS_TriggerStopRH.Q1 OR RS_TriggerStopCW.Q1) AND NOT bAutoCrossCut OR bTurretReturn AND bSafetyOK AND bTurretOverMedian AND IN_bTrtCrgReady AND IN_bTrtMOLReady AND NOT bTurretMedianRange AND NOT bAutoCrossCut AND NOT OUT_bCrgContactor AND OUT_bTrtContactor OR bMachineHoming AND bSafetyOK AND NOT bTurretReturn AND NOT bAutoCrossCut AND bCarriageHomeRH AND IN_bTrtCrgReady AND IN_bCrgMOLReady AND OUT_bCrgContactor AND NOT OUT_bTrtContactor;

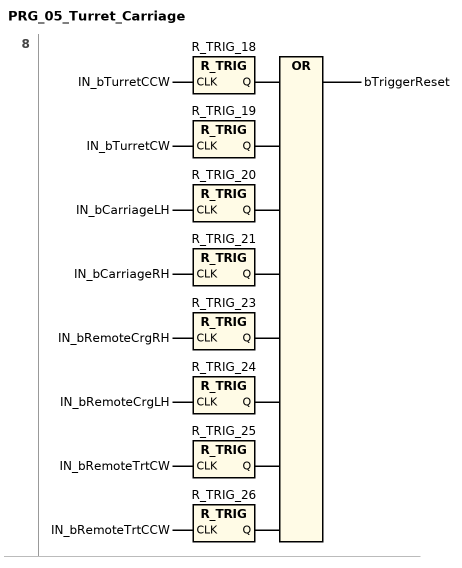
// NETWORK 8
R_TRIG_18(CLK := IN_bTurretCCW); // R_TRIG
R_TRIG_19(CLK := IN_bTurretCW); // R_TRIG
R_TRIG_20(CLK := IN_bCarriageLH); // R_TRIG
R_TRIG_21(CLK := IN_bCarriageRH); // R_TRIG
R_TRIG_23(CLK := IN_bRemoteCrgRH); // R_TRIG
R_TRIG_24(CLK := IN_bRemoteCrgLH); // R_TRIG
R_TRIG_25(CLK := IN_bRemoteTrtCW); // R_TRIG
R_TRIG_26(CLK := IN_bRemoteTrtCCW); // R_TRIG
bTriggerReset := R_TRIG_18.Q OR R_TRIG_19.Q OR R_TRIG_20.Q OR R_TRIG_21.Q OR R_TRIG_23.Q OR R_TRIG_24.Q OR R_TRIG_25.Q OR R_TRIG_26.Q;

END_PROGRAM

// ---- POUs/MAIN FUNCTIONS/PRG_06_HomePosition.TcPOU
PROGRAM PRG_06_HomePosition
VAR
	iStepHome: INT;
	SR_MachineHoming: SR;
	R_TRIG_MachineHoming: R_TRIG;	
	TON_HomingStep10: TON;
END_VAR

VAR PERSISTENT
	
END_VAR

	IF		NOT bSafetyOK OR IN_FaultReset OR bAutoCrossCut OR bTurretReturn OR NOT SR_MachineHoming.Q1
	THEN	iStepHome	:=	0;
			bMachineHoming := FALSE;
	END_IF
	
			R_TRIG_MachineHoming(	CLK:= IN_bLiftingPosition AND NOT bTurretReturn AND NOT bAutoCrossCut AND NOT OUT_bSawOn,
									Q=> );	
			SR_MachineHoming(	SET1:= R_TRIG_MachineHoming.Q AND NOT SR_MachineHoming.Q1,
								RESET:= (R_TRIG_MachineHoming.Q AND SR_MachineHoming.Q1) OR NOT bSafetyOK OR IN_FaultReset, 
								Q1=> );
	
IF bMachineHoming THEN
	OUT_bLiftingPositionLED := TRUE ;
ELSE
	OUT_bLiftingPositionLED := FALSE ;
END_IF

CASE iStepHome OF
	0:	// Init step
		bTurretHome		:= FALSE; 
	    bCarriageHomeLH	:= FALSE;
	    bCarriageHomeRH	:= FALSE;
	    bCrossCutHomeLH	:= FALSE;
	    bCrossCutHomeRH	:= FALSE;
		bZAxisHome := FALSE;
		TON_HomingStep10.IN := FALSE;
	
		IF R_TRIG_MachineHoming.Q AND bSafetyOK AND NOT OUT_bSawOn THEN
			bMachineHoming := TRUE ;
			iStepHome := 5 ;
		ELSE
			bMachineHoming := FALSE ;
		END_IF
		
	5:	// Raise Z-axis all the way up
	
		IF IN_bSawUpLimit AND bSafetyOK AND bMachineHoming THEN
			bZAxisHome := TRUE ;
		ELSE
			bZAxisHome := FALSE ; 
			iStepHome := 7 ;
		END_IF
		
	7:	// Move crosscut motor to centre
	 
		IF IN_uCrossCutSSI < (uRailLimitLeft + uRailLimitRight)/2 AND bSafetyOK AND bMachineHoming THEN
			bCrossCutHomeLH := TRUE ;
			bCrossCutHomeRH := FALSE ;
		ELSIF IN_uCrossCutSSI > (uRailLimitLeft + uRailLimitRight)/2 AND bSafetyOK AND bMachineHoming THEN
			bCrossCutHomeRH := TRUE ;
			bCrossCutHomeLH := FALSE ;
		ELSIF (IN_uCrossCutSSI > ((uRailLimitLeft + uRailLimitRight)/2) - 50) OR (IN_uCrossCutSSI < ((uRailLimitLeft + uRailLimitRight)/2) + 50) AND bSafetyOK AND bMachineHoming THEN
			bCrossCutHomeLH := FALSE ;
			bCrossCutHomeRH := FALSE ;
			iStepHome := 10 ;
		END_IF
	
	10:	// Rotate turret to max -90°
	
			TON_HomingStep10(IN:= , PT:= T#1S, Q=> , ET=> );
		IF NOT bTurretCCW AND bSafetyOK AND bMachineHoming THEN
			bTurretHome := TRUE ;
		ELSIF bTurretCCW AND bSafetyOK AND bMachineHoming THEN
			TON_HomingStep10.IN := TRUE ;
			bTurretHome := FALSE ;
			IF TON_HomingStep10.Q THEN
			    iStepHome := 20 ;
			END_IF
			
		END_IF
	
	20: // Offset carriage a little to the right		// 32.3 < CarriageHome < 32.5
	
		IF (fbCarriagePOS.Out.rScaled < 32.3) AND bMachineHoming AND bSafetyOK THEN
			bCarriageHomeRH := TRUE ;
			bCarriageHomeLH := FALSE ;
		ELSIF (fbCarriagePOS.Out.rScaled > 32.5) AND bMachineHoming AND bSafetyOK THEN
			bCarriageHomeLH := TRUE ;
			bCarriageHomeRH := FALSE ;
		ELSIF (fbCarriagePOS.Out.rScaled > 32.3) AND (fbCarriagePOS.Out.rScaled < 32.5) THEN
			bCarriageHomeRH := FALSE ;
			bCarriageHomeLH := FALSE ;
			iStepHome := 30 ;
		END_IF
	
	30: //Crosscut offset towards the control panel (CUT direction)		// 55.5 < CrosscutHome < 55.75
	
		IF (fbCrosscutSSI.Out.rScaled < 55.5) AND bMachineHoming AND bSafetyOK THEN
			bCrossCutHomeLH := TRUE ;
			bCrossCutHomeRH := FALSE ;
		ELSIF (fbCrosscutSSI.Out.rScaled > 55.75) AND bMachineHoming AND bSafetyOK THEN
			bCrossCutHomeRH := TRUE ;
			bCrossCutHomeLH := FALSE ;
		ELSIF (fbCrosscutSSI.Out.rScaled > 55.5) AND (fbCrosscutSSI.Out.rScaled < 55.75) THEN
			bCrossCutHomeLH := FALSE ;
			bCrossCutHomeRH := FALSE ;
			iStepHome := 0 ;
		END_IF
		
END_CASE

END_PROGRAM

// ---- POUs/MAIN FUNCTIONS/PRG_07_Servo.TcPOU
PROGRAM PRG_07_Servo
VAR
	fbMC_Power_Ax1: MC_Power;
	fbMC_Power_Ax2: MC_Power;
	fbMC_Jog_Ax1: MC_Jog;
	fbMC_Jog_Ax2: MC_Jog;
	fbMC_Reset_Ax1: MC_Reset;
	fbMC_Reset_Ax2: MC_Reset;
	fbMC_Stop_Ax1: MC_Stop;
	fbMC_Stop_Ax2: MC_Stop;
	
	rJogSpeed:	REAL;
	
	bTest1: BOOL;
	MC_ReadStatus_0: MC_ReadStatus;
	MC_ReadStatus_1: MC_ReadStatus;
	R_TRIG_0: R_TRIG;
	R_TRIG_1: R_TRIG;
	MC_MoveVelocity_0: MC_MoveVelocity;
	uAx1Encoder: UDINT;
	bJogSpeedChange: BOOL;
	t_JogSpeedChange: TP;
	JogSpeegTrig: F_TRIG;
	iPowerOverride: INT;
	tof_SawDownLimit: TOF;
	TRIG_SawDownLimit: r_trig;
	SR_SawDownLimit: SR;

	ton_SawDownLimitTimer: ton;
	SR_ZAxisBuffer: SR;
	F_TRIG_ZAxisCapturedValue: F_TRIG;
	rZAxisBufferSpeed: REAL;
	rZAxisSlowSpeed: REAL;
	rZAxisMedSpeed: REAL;
	rZAxisFastSpeed: REAL;
	sr_ZAxisBufferZone: SR;
	rZAxisCurrentFeedbackSpeed: REAL;
	F_TRIG_ZAxisUpperLimitValue: F_TRIG;
	F_TRIG_ZAxisLowerLimitValue: F_TRIG;
	iZAxisCapturedBufferValue: DINT;

END_VAR

ACTION ACT_07_1_Power:
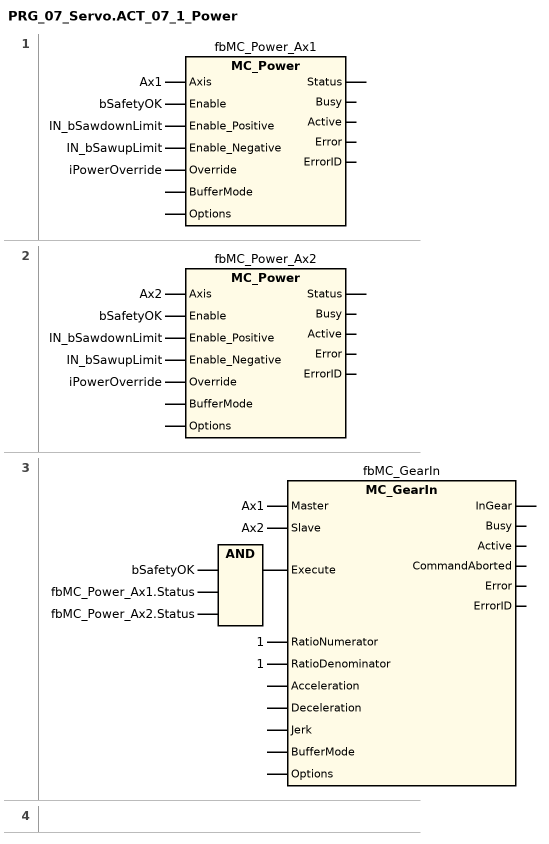
// NETWORK 1
fbMC_Power_Ax1(
    Axis := Ax1,
    Enable := bSafetyOK,
    Enable_Positive := IN_bSawdownLimit,
    Enable_Negative := IN_bSawupLimit,
    Override := iPowerOverride); // MC_Power

// NETWORK 2
fbMC_Power_Ax2(
    Axis := Ax2,
    Enable := bSafetyOK,
    Enable_Positive := IN_bSawdownLimit,
    Enable_Negative := IN_bSawupLimit,
    Override := iPowerOverride); // MC_Power

// NETWORK 3
fbMC_GearIn(
    Master := Ax1,
    Slave := Ax2,
    Execute := bSafetyOK AND fbMC_Power_Ax1.Status AND fbMC_Power_Ax2.Status,
    RatioNumerator := 1,
    RatioDenominator := 1); // MC_GearIn

// NETWORK 4
END_ACTION

ACTION ACT_07_2_Reset:
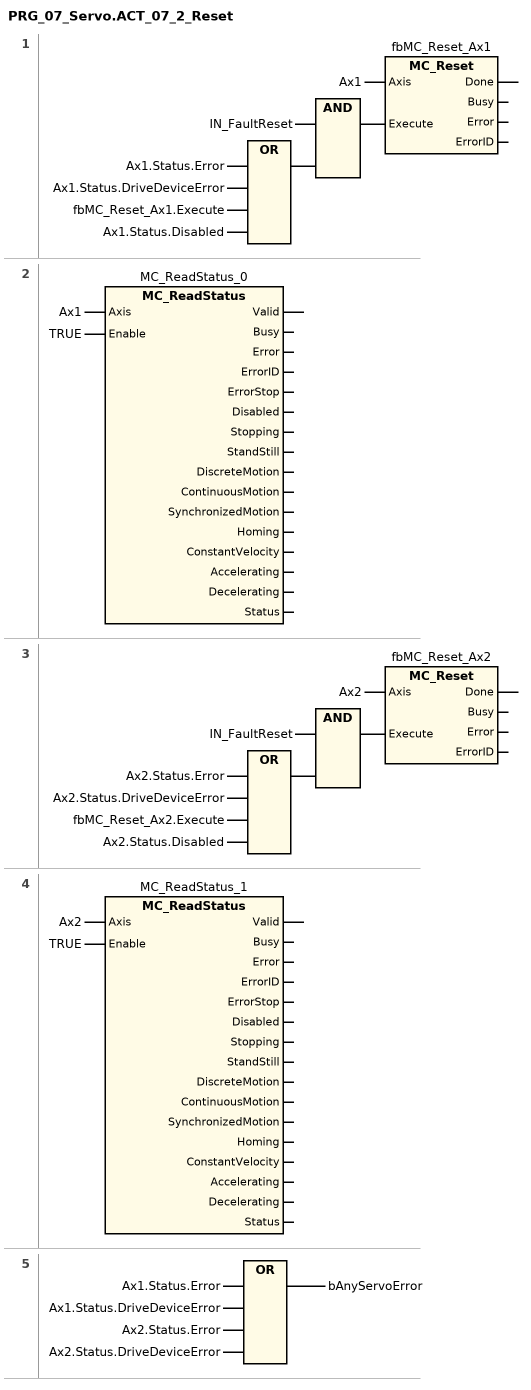
// NETWORK 1
fbMC_Reset_Ax1(Axis := Ax1, Execute := IN_FaultReset AND (Ax1.Status.Error OR Ax1.Status.DriveDeviceError OR fbMC_Reset_Ax1.Execute OR Ax1.Status.Disabled)); // MC_Reset

// NETWORK 2
MC_ReadStatus_0(Axis := Ax1, Enable := TRUE); // MC_ReadStatus

// NETWORK 3
fbMC_Reset_Ax2(Axis := Ax2, Execute := IN_FaultReset AND (Ax2.Status.Error OR Ax2.Status.DriveDeviceError OR fbMC_Reset_Ax2.Execute OR Ax2.Status.Disabled)); // MC_Reset

// NETWORK 4
MC_ReadStatus_1(Axis := Ax2, Enable := TRUE); // MC_ReadStatus

// NETWORK 5
bAnyServoError := Ax1.Status.Error OR Ax1.Status.DriveDeviceError OR Ax2.Status.Error OR Ax2.Status.DriveDeviceError;

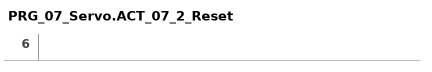
// NETWORK 6
END_ACTION

ACTION ACT_07_3_Jog:
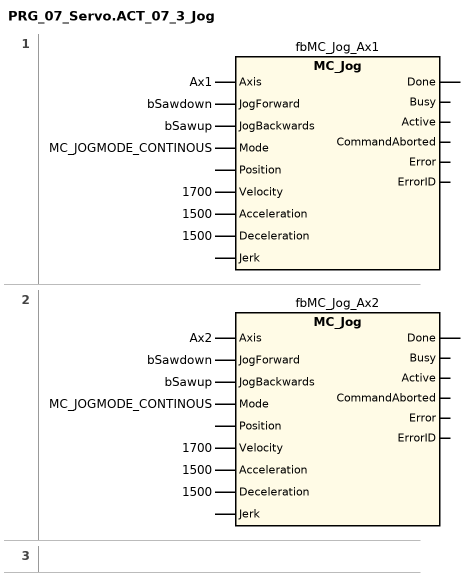
// NETWORK 1
fbMC_Jog_Ax1(
    Axis := Ax1,
    JogForward := bSawdown,
    JogBackwards := bSawup,
    Mode := MC_JOGMODE_CONTINOUS,
    Velocity := 1700,
    Acceleration := 1500,
    Deceleration := 1500); // MC_Jog

// NETWORK 2
fbMC_Jog_Ax2(
    Axis := Ax2,
    JogForward := bSawdown,
    JogBackwards := bSawup,
    Mode := MC_JOGMODE_CONTINOUS,
    Velocity := 1700,
    Acceleration := 1500,
    Deceleration := 1500); // MC_Jog

// NETWORK 3
END_ACTION

ACTION ACT_07_4_JogSpeed:
(* Z-axis speed setpoints *)
rZAxisBufferSpeed 	:= 950 ;
rZAxisSlowSpeed 	:= 1000 ;
rZAxisMedSpeed 		:= 1400 ;
rZAxisFastSpeed 	:= 1700 ;
rZAxisCurrentFeedbackSpeed := 750 ;

(* Z-axis capture value for the buffer zone *)
F_TRIG_ZAxisUpperLimitValue(CLK:= IN_bSawUpLimit, Q=> );
IF bSawUP AND F_TRIG_ZAxisUpperLimitValue.Q THEN
	iZAxisUpperLimitValue := LREAL_TO_DINT(Ax1.NcToPlc.ActPos) ;
END_IF

F_TRIG_ZAxisLowerLimitValue(CLK:= IN_bSawDownLimit, Q=> );
IF F_TRIG_ZAxisLowerLimitValue.Q THEN
	iZAxisLowerLimitValue := LREAL_TO_DINT(Ax1.NcToPlc.ActPos) ;
END_IF

	iZAxisCapturedBufferValue := iZAxisLowerLimitValue - 17040 ;	// approx. 3" high from the bed

(* Z-axis selector switch *)
IF		IN_bZaxisSlow	THEN
		rJogSpeed	:=	rZAxisSlowSpeed	;
ELSIF	IN_bZaxisFAST	THEN
		rJogSpeed	:=	rZAxisFastSpeed	;
ELSE	rJogSpeed	:=	rZAxisMedSpeed	;
END_IF

(* Z-axis power override limit at max 100% and min 0% *)
IF iPowerOverride > 100 THEN
	iPowerOverride := 100 ;
ELSIF iPowerOverride < 0 THEN
	iPowerOverride := 0 ;
END_IF

 (* Z-axis Jog speed *)
IF (Ax1.NcToPlc.ActPos > DINT_TO_LREAL(iZAxisCapturedBufferValue)) AND bSawDOWN AND rCrossCutSpeedMultiplier > 0.75 THEN	
	iPowerOverride := REAL_TO_INT((rZAxisBufferSpeed / rZAxisFastSpeed)*100) ;			// Z-axis buffer zone speed
	
ELSIF bSawDOWN AND rCrossCutSpeedMultiplier <= 0.75 THEN	
	iPowerOverride := REAL_TO_INT((rZAxisCurrentFeedbackSpeed / rZAxisFastSpeed)*100) ;	// Z-axis current feedback speed
	
ELSIF (Ax1.NcToPlc.ActPos >= DINT_TO_LREAL(iZAxisCapturedBufferValue)) AND bSawDOWN AND rCrossCutSpeedMultiplier > 0.75 THEN
	iPowerOverride := REAL_TO_INT((rJogSpeed / rZAxisFastSpeed)*100) ;					// Z-axis speed selector switch
	
ELSIF NOT bSawDOWN OR bSawUP THEN
	iPowerOverride := 100 ;
END_IF
END_ACTION

ACTION ACT_07_5_Stop:
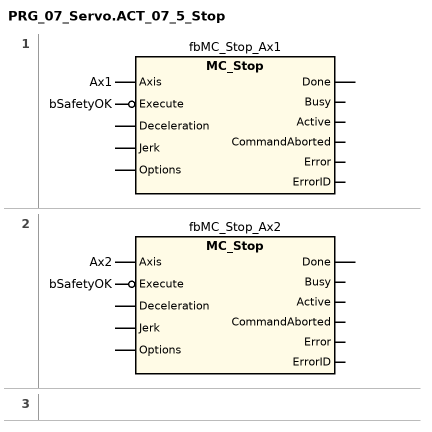
// NETWORK 1
fbMC_Stop_Ax1(Axis := Ax1, Execute := NOT bSafetyOK); // MC_Stop

// NETWORK 2
fbMC_Stop_Ax2(Axis := Ax2, Execute := NOT bSafetyOK); // MC_Stop

// NETWORK 3
END_ACTION

END_PROGRAM

// ---- POUs/MAIN FUNCTIONS/PRG_08_AnalogSignal.TcPOU
PROGRAM PRG_08_AnalogSignal
VAR
	uTurretValue: UDINT;
	iTRTEncoderValue: INT;
	TON_TeachLimit: TON;
	R_TRIG_TeachLimit: R_TRIG;
	RS_TurretBuffer: RS;
	R_TRIG_TurretBufferTrig: R_TRIG;
	F_TRIG_CarriageMedian: F_TRIG;
	TP_CarriageCaptureMedian: TP;
	F_TRIG_CarriageCaptureMedian: F_TRIG;
	F_TRIG_CarriageLeft: F_TRIG;
	TP_CarriageCaptureLeft: TP;
	F_TRIG_CarriageCaptureLeft: F_TRIG;
	F_TRIG_CarriageRight: F_TRIG;
	TP_CarriageCaptureRight: TP;
	F_TRIG_CarriageCaptureRight: F_TRIG;

	iCarriageAbsoluteMedian: INT;
	rCrossCutOffset: REAL;
	uCrossCutMax: UDINT;
	uCrossCutMin: UDINT;
	rRailHypotenuse: LREAL;
	iRailHypotenuse: UINT;
	uTeachLimit: UINT;
	rCarriageOffsetMultiplier: LREAL;
	rTurretOffsetMultiplier: LREAL;
	rCarriageVariable: LREAL;
	rTurretVariable: LREAL;
	iOffsetStep: INT;
	rCosineAngle: REAL;
	rConvertedOffset: REAL;
	iRailHypotenuseLeft: UINT;
	iRailHypotenuseRight: UINT;
	rAddend: REAL;
	R_TRIG_TurretValue: R_TRIG;
	
	bTurretEncoderCW: BOOL;
	bTurretEncoderCCW: BOOL;
	uTurretEncoderAddedValue: UDINT;
	
END_VAR

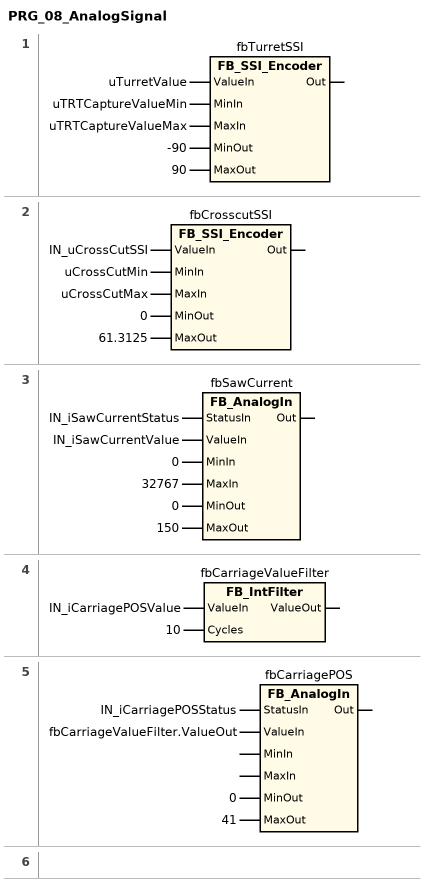
// NETWORK 1
fbTurretSSI(
    ValueIn := uTurretValue,
    MinIn := uTRTCaptureValueMin,
    MaxIn := uTRTCaptureValueMax,
    MinOut := -90,
    MaxOut := 90); // FB_SSI_Encoder

// NETWORK 2
fbCrosscutSSI(
    ValueIn := IN_uCrossCutSSI,
    MinIn := uCrossCutMin,
    MaxIn := uCrossCutMax,
    MinOut := 0,
    MaxOut := 61.3125); // FB_SSI_Encoder

// NETWORK 3
fbSawCurrent(
    StatusIn := IN_iSawCurrentStatus,
    ValueIn := IN_iSawCurrentValue,
    MinIn := 0,
    MaxIn := 32767,
    MinOut := 0,
    MaxOut := 150); // FB_AnalogIn

// NETWORK 4
fbCarriageValueFilter(ValueIn := IN_iCarriagePOSValue, Cycles := 10); // FB_IntFilter

// NETWORK 5
fbCarriagePOS(
    StatusIn := IN_iCarriagePOSStatus,
    ValueIn := fbCarriageValueFilter.ValueOut,
    MinOut := 0,
    MaxOut := 41); // FB_AnalogIn

// NETWORK 6

ACTION ACT_08_1_TurretSSI:
(* ########### ABSOLUTE 0 DEGREES: IN_uTurretSSI = 16238 @ SSI Data length of 15 ##################### *)
(* SSI Data length: 0x000F(15) *)

(* Turret Median, Max, Min *)
R_TRIG_TurretValue(CLK:= IN_bTurretRotationReference, Q=> );

	uTurretSSIMedian := 3188 + 32767 ;	// AP2 Turret median = 3188

	// Capture Min value and trigger stop at max CW
IF(* NOT *)IN_bTurretRotationReference AND (fbTurretSSI.Out.rScaled < -85) AND (IN_bTurretCW OR IN_bRemoteTrtCW) THEN
	uTRTCaptureValueMin := IN_uTurretSSI + 32767 - uTurretEncoderAddedValue ;		// Temp Min 21643
	bTurretMedian := FALSE ;
	bTurretCW := TRUE ;
	bTurretCCW := FALSE ;
	
	// Trigger stop at CW in case turret rotates past min value
ELSIF (uTRTCaptureValueMin <= uTRTCaptureValueMin - 50)	   THEN
	bTurretMedian := FALSE ;
	bTurretCW := TRUE ;
	bTurretCCW := FALSE ;

	// Capture Max value and trigger stop at max CCW
ELSIF ((* NOT *) IN_bTurretRotationReference AND (fbTurretSSI.Out.rScaled > 85) AND (IN_bTurretCCW OR IN_bRemoteTrtCCW)) OR
		((* NOT *) IN_bTurretRotationReference AND bTurretHome AND fbTurretSSI.Out.rScaled > 85) THEN
	uTRTCaptureValueMax := IN_uTurretSSI + 32767 - uTurretEncoderAddedValue ;		// Temp Max 50267
	bTurretMedian := FALSE ;
	bTurretCW := FALSE ;
	bTurretCCW := TRUE ;
	
	// Trigger stop at CCW in case turret rotates past max value
ELSIF (uTRTCaptureValueMax >= uTRTCaptureValueMax + 50)	  THEN
	bTurretMedian := FALSE ;
	bTurretCW := FALSE ;
	bTurretCCW := TRUE ;
	
	// Limits are off when Turret reference limit switch is triggered
ELSIF R_TRIG_TurretValue.Q AND  (fbTurretSSI.Out.rScaled > 85) THEN
	bTurretMedian := FALSE ;
	bTurretCW := FALSE ;
	bTurretCCW := FALSE ;
	
	// Limits are off when Turret reference limit switch is triggered
ELSIF R_TRIG_TurretValue.Q AND  (fbTurretSSI.Out.rScaled < -85) THEN
	bTurretMedian := FALSE ;
	bTurretCW := FALSE ;
	bTurretCCW := FALSE ;
	
END_IF

(* Turret rollover range *)		(* clockwise rollover, encoder value going down *)
IF ((IN_uTurretSSI <= 32767) AND (IN_uTurretSSI >= 20500)) THEN		// ########### dependent on range of encoder rollover #######################
	bTurretEncoderCW := TRUE ;
	uTurretEncoderAddedValue := 32767 ;
ELSE
	bTurretEncoderCW   := FALSE ;
	uTurretEncoderAddedValue := 0 ;
END_IF

(* Turret value going past min and max *)
IF (IN_uTurretSSI + 32767 - uTurretEncoderAddedValue < uTRTCaptureValueMax) AND (IN_uTurretSSI + 32767 - uTurretEncoderAddedValue > uTRTCaptureValueMin) THEN
	uTurretValue := IN_uTurretSSI + 32767 - uTurretEncoderAddedValue ;	
ELSIF (IN_uTurretSSI + 32767 - uTurretEncoderAddedValue > uTRTCaptureValueMax) THEN
	uTurretValue := uTRTCaptureValueMax ;
ELSIF (IN_uTurretSSI + 32767 - uTurretEncoderAddedValue < uTRTCaptureValueMin) THEN
	uTurretValue := uTRTCaptureValueMin ;
END_IF

(* Trigger stop turret at 0° *)
IF (IN_uTurretSSI + 32767 - uTurretEncoderAddedValue >= (uTurretSSIMedian-1)) AND (IN_uTurretSSI + 32767 - uTurretEncoderAddedValue <= (uTurretSSIMedian+1)) THEN
	bTurretMedianRange := TRUE;
ELSE bTurretMedianRange := FALSE;
END_IF 

(* ######################### NEW ############################# *)
(* Turret 0° - 45° range *)
IF fbTurretSSI.Out.rScaled > -47 AND fbTurretSSI.Out.rScaled < 47 THEN
	bTurret045Range := TRUE ;
ELSE bTurret045Range := FALSE ;
END_IF
(* ######################### NEW ############################# *)

(* Turret Encoder Display *)
(* (ValueIN/MaxIN)*32767  *)
OUT_iEncoderDisplay := iTRTEncoderValue ;
iTRTEncoderValue := REAL_TO_INT((((UDINT_TO_REAL(IN_uTurretSSI + 32767 - uTurretEncoderAddedValue - uTRTCaptureValueMin)) / UDINT_TO_REAL(uTRTCaptureValueMax - uTRTCaptureValueMin))*32767 ));
IF ((iTRTEncoderValue < 0) AND bTurretOverMedian) OR ((IN_uTurretSSI + 32767 - uTurretEncoderAddedValue > uTRTCaptureValueMax) AND bTurretOverMedian) THEN
	iTRTEncoderValue := 32767 ;
ELSIF ((iTRTEncoderValue < 0) AND bTurretUnderMedian) OR ((IN_uTurretSSI + 32767 - uTurretEncoderAddedValue < uTRTCaptureValueMin) AND bTurretUnderMedian) THEN
	iTRTEncoderValue := 0 ;
END_IF

(* Turret Return variable *)
IF (IN_uTurretSSI + 32767 - uTurretEncoderAddedValue > uTurretSSIMedian) AND NOT bTurretMedianRange THEN
	bTurretOverMedian := TRUE;
ELSE 	bTurretOverMedian := FALSE;
END_IF

IF (IN_uTurretSSI + 32767 - uTurretEncoderAddedValue < uTurretSSIMedian) AND NOT bTurretMedianRange THEN
	bTurretUnderMedian := TRUE;
ELSE 	bTurretUnderMedian := FALSE;
END_IF

(* Buffer zone for turret to slow down before approaching the trigger points at 0°, 90°, and -90° *)
R_TRIG_TurretBufferTrig(CLK:= bTurretMedianRange, Q=> );
RS_TurretBuffer(SET:= R_TRIG_TurretBufferTrig.Q, 
				RESET1:=  (IN_bTurretCCW OR IN_bRemoteTrtCCW OR IN_bTurretCW OR IN_bRemoteTrtCW), 
				Q1=> );

IF ((IN_uTurretSSI + 32767 - uTurretEncoderAddedValue >= (uTurretSSIMedian-100)) AND NOT (IN_uTurretSSI + 32767 - uTurretEncoderAddedValue >= uTurretSSIMedian) AND (IN_bTurretCCW OR IN_bRemoteTrtCCW OR (bTurretReturn AND OUT_bTrtCrgLH))) OR
	((IN_uTurretSSI + 32767 - uTurretEncoderAddedValue <= (uTurretSSIMedian+100)) AND NOT (IN_uTurretSSI + 32767 - uTurretEncoderAddedValue <= uTurretSSIMedian) AND (IN_bTurretCW OR IN_bRemoteTrtCW OR (bTurretReturn AND OUT_bTrtCrgRH))) OR
	((IN_uTurretSSI + 32767 - uTurretEncoderAddedValue <= (uTRTCaptureValueMin+100)) AND (IN_bTurretCW OR IN_bRemoteTrtCW OR (bTurretReturn AND OUT_bTrtCrgRH) OR bMachineHoming)) OR
	((IN_uTurretSSI + 32767 - uTurretEncoderAddedValue >= (uTRTCaptureValueMax-100)) AND (IN_bTurretCCW OR IN_bRemoteTrtCCW OR (bTurretReturn AND OUT_bTrtCrgLH) OR bMachineHoming))
THEN
	bTurretBufferSpeed := TRUE;
ELSE
	bTurretBufferSpeed := FALSE;
END_IF
END_ACTION

ACTION ACT_08_2_CrossCutSSI:
(* SSI Data length: 0x000F(15) *)
(* encoder values *)
uRailLimitLeft := 16210 ;//3746 ;	// align centre of the blade with the left inner edge of the bed rails
uRailLimitRight := 14953 ;//2625 ;	// align centre of the blade with the right inner edge of the bed rails
uCrossCutMax := 16356 ;//3893 ;		// move the saw block all the way to the left
uCrossCutMin := 15099 ;//2480 ;		// move the saw block all the way to the right

(* CrossCut Limits *)
IF (IN_uCrossCutSSI+32767 <= (uCrossCutMedian - (iRailHypotenuse - uTeachLimit))+32767) OR
	(((fbTurretSSI.Out.rScaled > 85 (*Degrees*)) OR (fbTurretSSI.Out.rScaled < -85)) AND (fbCrosscutSSI.Out.rScaled <= (fbCrosscutSSI.MinOut + 6 (*Inches*)))) OR
	(IN_uCrossCutSSI < (uCrossCutMin + 2))
	THEN
	bLimitRight := TRUE ;
	bLimitLeft := FALSE ;
ELSIF (IN_uCrossCutSSI+32767 >= (uCrossCutMedian + (iRailHypotenuse - uTeachLimit))+32767) OR
	(((fbTurretSSI.Out.rScaled > 85 (*Degrees*)) OR (fbTurretSSI.Out.rScaled < -85)) AND (fbCrosscutSSI.Out.rScaled >= (fbCrosscutSSI.MaxOut - 6 (*Inches*)))) OR
	(IN_uCrossCutSSI > (uCrossCutMax - 2))
	THEN
	bLimitLeft := TRUE ;
	bLimitRight := FALSE ;
ELSE
	bLimitRight := FALSE ;
	bLimitLeft 	:= FALSE ;
END_IF

(* Approaching Limits for Crosscut buffer zone *)
IF (IN_uCrossCutSSI+32767 <= (uCrossCutMedian - (iRailHypotenuse - uTeachLimit))+50+32767) OR 
	(((fbTurretSSI.Out.rScaled > 85 (*Degrees*)) OR (fbTurretSSI.Out.rScaled < -85)) AND (fbCrosscutSSI.Out.rScaled <= (fbCrosscutSSI.MinOut + 6)+1)) OR
	(IN_uCrossCutSSI <= (uCrossCutMin + 50))
	THEN
	bApproachingLimitRight := TRUE ;
	bApproachingLimitLeft := FALSE ;
ELSIF (IN_uCrossCutSSI+32767 >= (uCrossCutMedian + (iRailHypotenuse - uTeachLimit))-50+32767) OR 
	(((fbTurretSSI.Out.rScaled > 85 (*Degrees*)) OR (fbTurretSSI.Out.rScaled < -85)) AND (fbCrosscutSSI.Out.rScaled >= (fbCrosscutSSI.MaxOut - 6)-1))  OR
	(IN_uCrossCutSSI >= (uCrossCutMax - 50))
	THEN
	bApproachingLimitLeft := TRUE ;
	bApproachingLimitRight := FALSE ;
ELSE
	bApproachingLimitRight := FALSE ;
	bApproachingLimitLeft 	:= FALSE ;
END_IF

(*	bApproachingLimitRight := FALSE ;
	bApproachingLimitLeft 	:= FALSE ;
	bLimitRight := FALSE ;
	bLimitLeft 	:= FALSE ;
*)
(* Hypotenuse calculation *)
IF ABS(fbTurretSSI.Out.rScaled) <> 90 THEN
	rCosineAngle := COS ( (PI / 180) * ABS( fbTurretSSI.Out.rScaled)) ;
ELSE
	rCosineAngle := COS ( (PI / 180) * 89.9999 ) ;
END_IF

uTeachLimit := REAL_TO_UINT(((UDINT_TO_REAL(uRailLimitLeft - uRailLimitRight))/2) - ((UDINT_TO_REAL(uTeachLimitLeft - uTeachLimitRight))/2)) ;

fbTurretSSI.Out.rScaled ; // Turret Angle

	rRailHypotenuse := ( (UDINT_TO_LREAL(uRailLimitLeft - uRailLimitRight)/2) / rCosineAngle);
	
//	iRailHypotenuse := LREAL_TO_UINT(rRailHypotenuse);
IF rRailHypotenuse >= 6436 OR rRailHypotenuse < 0 THEN
	iRailHypotenuse := 6436;		// rRailHypotenuse = 6436 	@ 85°
ELSE
	iRailHypotenuse := LREAL_TO_UINT(rRailHypotenuse);
END_IF

(* Carriage Position Offset *)
fbCarriagePOS.Out.rScaled;
fbCrosscutSSI.Out.rScaled;

F_TRIG_CarriageMedian(CLK:= IN_bCarriageReference, Q=> );
TP_CarriageCaptureMedian(IN:= F_TRIG_CarriageMedian.Q, PT:= T#0.5S, Q=> , ET=> );
F_TRIG_CarriageCaptureMedian(CLK:= TP_CarriageCaptureMedian.Q, Q=> );
IF F_TRIG_CarriageCaptureMedian.Q THEN		
	iCarriageMedian := fbCarriageValueFilter.ValueOut ;
END_IF

iOffsetStep;
IF NOT IN_bCarriageReference THEN
	rCrossCutOffset := 0 ;
ELSE
	rCrossCutOffset := ABS(fbCarriagePOS.Out.rScaled - ((fbCarriagePOS.MaxOut-fbCarriagePOS.MinOut)/2)) + rAddend ;
		IF 		IN_bCarriageReference AND NOT bTurretMedianRange AND (fbCarriageValueFilter.ValueOut < iCarriageMedian AND fbTurretSSI.Out.rScaled > 55) THEN
			rAddend := 0.75 ; iOffsetStep := 1;	// Carriage left, Turret CCW
		ELSIF	IN_bCarriageReference AND NOT bTurretMedianRange AND (fbCarriageValueFilter.ValueOut > iCarriageMedian AND fbTurretSSI.Out.rScaled > 55) THEN
			rAddend := 0 ; iOffsetStep := 2;	// Carriage right, Turret CCW
		ELSIF	IN_bCarriageReference AND NOT bTurretMedianRange AND (fbCarriageValueFilter.ValueOut > iCarriageMedian AND fbTurretSSI.Out.rScaled < -55) THEN
			rAddend := 0.5 ; iOffsetStep := 3;	// Carriage right, Turret CW
		ELSIF	IN_bCarriageReference AND NOT bTurretMedianRange AND (fbCarriageValueFilter.ValueOut < iCarriageMedian AND fbTurretSSI.Out.rScaled < -55) THEN
			rAddend := 0 ; iOffsetStep := 4;	// Carriage left, Turret CW
		ELSE
			rAddend := 0 ; iOffsetStep := 10;
		END_IF
END_IF

(* Crosscut median *)
rTurretOffsetMultiplier := (rTurretVariable * (ABS(fbTurretSSI.Out.rScaled)/90)) ;

IF (NOT IN_bCarriageReference AND fbTurretSSI.Out.rScaled >0) OR (IN_bCarriageReference AND (fbTurretSSI.Out.rScaled > 85 OR fbTurretSSI.Out.rScaled < -85)) THEN	
	uCrossCutMedian := REAL_TO_UDINT (((UDINT_TO_REAL(uTeachLimitLeft + uTeachLimitRight)) / 2 ) -  ((rTurretOffsetMultiplier/(fbCrosscutSSI.MaxOut-fbCrosscutSSI.MinOut))*UDINT_TO_REAL(uCrossCutMax-uCrossCutMin))  ) ;
	rTurretVariable := 0.5;
ELSIF (NOT IN_bCarriageReference AND fbTurretSSI.Out.rScaled <0) OR (IN_bCarriageReference AND (fbTurretSSI.Out.rScaled > 85 OR fbTurretSSI.Out.rScaled < -85)) THEN	
	uCrossCutMedian := REAL_TO_UDINT (((UDINT_TO_REAL(uTeachLimitLeft + uTeachLimitRight)) / 2 ) +  ((rTurretOffsetMultiplier/(fbCrosscutSSI.MaxOut-fbCrosscutSSI.MinOut))*UDINT_TO_REAL(uCrossCutMax-uCrossCutMin))  ) ;
	rTurretVariable := 0.5;
ELSIF IN_bCarriageReference AND (fbCarriageValueFilter.ValueOut < iCarriageMedian) AND NOT (fbTurretSSI.Out.rScaled > 85 OR fbTurretSSI.Out.rScaled < -85) THEN
	uCrossCutMedian := REAL_TO_UDINT(((UDINT_TO_REAL(uTeachLimitLeft + uTeachLimitRight)) / 2 ) - ((rCrossCutOffset/(fbCrosscutSSI.MaxOut-fbCrosscutSSI.MinOut))*UDINT_TO_REAL(uCrossCutMax-uCrossCutMin)) /rCosineAngle) ;
ELSIF IN_bCarriageReference AND (fbCarriageValueFilter.ValueOut > iCarriageMedian) AND NOT (fbTurretSSI.Out.rScaled > 85 OR fbTurretSSI.Out.rScaled < -85) THEN
	uCrossCutMedian := REAL_TO_UDINT(((UDINT_TO_REAL(uTeachLimitLeft + uTeachLimitRight)) / 2 ) + ((rCrossCutOffset/(fbCrosscutSSI.MaxOut-fbCrosscutSSI.MinOut))*UDINT_TO_REAL(uCrossCutMax-uCrossCutMin)) /rCosineAngle) ;
END_IF

IF (IN_uCrossCutSSI >= (uCrossCutMedian - 10)) AND (IN_uCrossCutSSI <= (uCrossCutMedian + 10)) THEN
	bCrossCutCentre := TRUE ;
ELSE
	bCrossCutCentre := FALSE ;
END_IF
(* ################################################# REMOVE AFTER SETUP ########################
IF (IN_uCrossCutSSI >= (uCrossCutMedian - 30)) AND (IN_uCrossCutSSI <= (uCrossCutMedian + 30)) THEN
	bCrossCutCentreForRotation := TRUE ;
ELSE
	bCrossCutCentreForRotation := FALSE ;
END_IF
################################################# REMOVE AFTER SETUP ######################## *)
	bCrossCutCentreForRotation := TRUE ;

(* Teach Limits left and right *)
TON_TeachLimit(IN:= (IN_bTeach AND ((IN_bTeachLeft AND IN_uCrossCutSSI > (uCrossCutMedian+100)) OR (IN_bTeachRight AND IN_uCrossCutSSI < (uCrossCutMedian-100))) AND NOT IN_bCarriageReference AND bTurretMedianRange AND NOT (bTurretReturn OR bAutoCrossCut OR bMachineHoming OR OUT_bSawON)),
				PT:= T#3S, Q=> , ET=> );
OUT_bTeachLED := NOT TON_TeachLimit.Q AND IN_bTeach AND NOT IN_bCarriageReference AND bTurretMedianRange AND ((IN_bTeachLeft AND IN_uCrossCutSSI > (uCrossCutMedian+100)) OR (IN_bTeachRight AND IN_uCrossCutSSI < (uCrossCutMedian-100))) ;
R_TRIG_TeachLimit(CLK:= TON_TeachLimit.Q, Q=> );

IF NOT IN_bCarriageReference AND R_TRIG_TeachLimit.Q AND IN_bTeachLeft AND bTurretMedianRange AND NOT (bTurretReturn AND bAutoCrossCut AND bMachineHoming) THEN
	uTeachLimitLeft := IN_uCrossCutSSI;
ELSIF NOT IN_bCarriageReference AND R_TRIG_TeachLimit.Q AND IN_bTeachRight AND bTurretMedianRange AND NOT (bTurretReturn AND bAutoCrossCut AND bMachineHoming) THEN
	uTeachLimitRight := IN_uCrossCutSSI;
END_IF

(* crash positions *)
IF 		(fbCarriagePOS.Out.rScaled <= 24 AND fbTurretSSI.Out.rScaled >= 50 AND fbCrosscutSSI.Out.rScaled >= 46) 	// echain @ corner #1
	OR 	(fbCarriagePOS.Out.rScaled <= 41 AND fbTurretSSI.Out.rScaled >= 70 AND fbCrosscutSSI.Out.rScaled >= 57)		// light bar @ side 1-2
	OR	(fbCarriagePOS.Out.rScaled <= 30 AND fbTurretSSI.Out.rScaled <= -65 AND fbCrosscutSSI.Out.rScaled >= 59)	// corner 4
	OR	(fbCarriagePOS.Out.rScaled <= 30 AND fbTurretSSI.Out.rScaled >= 60 AND fbCrosscutSSI.Out.rScaled >= 51)		// echain @ corner #1
	OR	(fbCarriagePOS.Out.rScaled >= 36 AND fbTurretSSI.Out.rScaled <= -60 AND fbCrosscutSSI.Out.rScaled >= 60)	// corner 4
	OR	(fbCarriagePOS.Out.rScaled >= 30 AND fbTurretSSI.Out.rScaled <= -50 AND fbCrosscutSSI.Out.rScaled >= 57.5)	// corner 4
THEN
	bEchainCrashPosLeft := TRUE ;		// Crosscut Left limit
	bEchainCrashPosRight := FALSE ;
ELSIF 	(fbCarriagePOS.Out.rScaled <= 14 AND fbTurretSSI.Out.rScaled <= -85 AND fbCrosscutSSI.Out.rScaled <= 15) 	// echain @ corner #1
	OR	(fbCarriagePOS.Out.rScaled <= 17.5 AND fbTurretSSI.Out.rScaled >= 75 AND fbCrosscutSSI.Out.rScaled <= 10.5)	// echain @ corner #3
	OR  (fbCarriagePOS.Out.rScaled <= 30 AND fbTurretSSI.Out.rScaled <= -65 AND fbCrosscutSSI.Out.rScaled <= 7)		// light bar @ side 1-2
	OR  (fbCarriagePOS.Out.rScaled <= 10 AND fbTurretSSI.Out.rScaled <= -70 AND fbCrosscutSSI.Out.rScaled <= 16)	// echain @ corner #1
	OR  (fbCarriagePOS.Out.rScaled >= 21 AND fbTurretSSI.Out.rScaled >= 60 AND fbCrosscutSSI.Out.rScaled <= 7)		// corner #4
	OR  (fbCarriagePOS.Out.rScaled <= 21 AND fbTurretSSI.Out.rScaled >= 60 AND fbCrosscutSSI.Out.rScaled <= 7)		// servomotor side #3-4
	OR  (fbCarriagePOS.Out.rScaled <= 16 AND fbTurretSSI.Out.rScaled >= 60 AND fbCrosscutSSI.Out.rScaled <= 17)		// horizontal echain @ corner #3
	OR  (fbCarriagePOS.Out.rScaled >= 16 AND fbTurretSSI.Out.rScaled >= 65 AND fbCrosscutSSI.Out.rScaled <= 5)		// spray bar side #3-4
THEN
	bEchainCrashPosLeft := FALSE ;		// Crosscut Right limit
	bEchainCrashPosRight := TRUE ;
ELSE
	bEchainCrashPosLeft := FALSE ;
	bEchainCrashPosRight := FALSE ;
END_IF
END_ACTION

ACTION ACT_08_3_CarriagePOS:
(* Carriage end limits *)
F_TRIG_CarriageLeft(CLK:= IN_bCarriageLHLimit, Q=> );
TP_CarriageCaptureLeft(IN:= F_TRIG_CarriageLeft.Q, PT:= T#0.5S, Q=> , ET=> );
F_TRIG_CarriageCaptureLeft(CLK:= TP_CarriageCaptureLeft.Q, Q=> );
IF F_TRIG_CarriageCaptureLeft.Q THEN
	iCarriageLeftLimit := fbCarriageValueFilter.ValueOut ;
END_IF

IF fbCarriageValueFilter.ValueOut >= iCarriageLeftLimit THEN
	fbCarriagePOS.MinIn := iCarriageLeftLimit ;
ELSIF fbCarriageValueFilter.ValueOut < iCarriageLeftLimit THEN
	fbCarriagePOS.MinIn := fbCarriageValueFilter.ValueOut ;
END_IF


F_TRIG_CarriageRight(CLK:= IN_bCarriageRHLimit, Q=> );
TP_CarriageCaptureRight(IN:= F_TRIG_CarriageRight.Q, PT:= T#0.5S, Q=> , ET=> );
F_TRIG_CarriageCaptureRight(CLK:= TP_CarriageCaptureRight.Q, Q=> );
IF F_TRIG_CarriageCaptureRight.Q THEN
	iCarriageRightLimit := fbCarriageValueFilter.ValueOut ;
END_IF

IF fbCarriageValueFilter.ValueOut <= iCarriageRightLimit THEN
	fbCarriagePOS.MaxIn := iCarriageRightLimit ;
ELSIF fbCarriageValueFilter.ValueOut > iCarriageRightLimit THEN
	fbCarriagePOS.MaxIn := fbCarriageValueFilter.ValueOut ;
END_IF

iCarriageAbsoluteMedian := ( iCarriageRightLimit + iCarriageLeftLimit ) / 2 ;
END_ACTION

END_PROGRAM

// ---- POUs/FUNCTION BLOCKS/FB_SSI_Encoder.TcPOU
FUNCTION_BLOCK FB_SSI_Encoder
VAR_INPUT
	
	ValueIn		: UDINT;				(* Analog input value *)
	MinIn		: UDINT;				(* Minimum value for input signal *)
	MaxIn		: UDINT;				(* Maximum value for input signal *)
	MinOut		: REAL;					(* Minimum value for output signal *)
	MaxOut		: REAL;					(* Maximum value for output signal *)
	
END_VAR
VAR_OUTPUT
	Out			: SSI_Encoder ;
END_VAR
VAR
	RangeIn: REAL;
	RangeOut: REAL;
END_VAR

(* Rescale input *)

	RangeIn 			:= UDINT_TO_REAL( MaxIn ) - UDINT_TO_REAL( MinIn );

	RangeOut 			:= MaxOut - MinOut;

	IF RangeIn <> 0
	(*  AND ValueIn >= MinIn
	  AND ValueIn <= MaxIn *) THEN
		Out.rScaled 	:= ( ( ( UDINT_TO_REAL( ValueIn  -  MinIn ) ) / RangeIn ) * RangeOut ) + MinOut;
	ELSE
		Out.rScaled		:= 0;
	END_IF

	Out.uCounterValue			:= ValueIn;

END_FUNCTION_BLOCK

// ---- POUs/FUNCTION BLOCKS/FB_AnalogIn.TcPOU
FUNCTION_BLOCK FB_AnalogIn
VAR_INPUT
	StatusIn	: INT;					(* Status Analog input signal *)
	ValueIn		: INT;					(* Analog input value *)
	MinIn		: INT;					(* Minimum value for input signal *)
	MaxIn		: INT;					(* Maximum value for input signal *)
	MinOut		: REAL;					(* Minimum value for output signal *)
	MaxOut		: REAL;					(* Maximum value for output signal *)
END_VAR
VAR
	RangeIn		: REAL;
	RangeOut	: REAL;
END_VAR
VAR_OUTPUT
	Out			: AnalogSignal;
END_VAR

(* Rescale Input *)
	RangeIn 			:= INT_TO_REAL( MaxIn ) - INT_TO_REAL( MinIn );

	RangeOut 			:= MaxOut - MinOut;

	IF RangeIn <> 0
	  AND ValueIn >= MinIn
	  AND ValueIn <= MaxIn THEN
		Out.rScaled 	:= ( ( ( INT_TO_REAL( ValueIn ) - INT_TO_REAL( MinIn ) ) / RangeIn ) * RangeOut ) + MinOut;
	ELSE
		Out.rScaled		:= 0;
	END_IF

	Out.iRawVal			:= ValueIn;

(* Status *)
	Out.bUnderRange 	:= StatusIn.0;
	Out.bOverRange 		:= StatusIn.1;
	Out.bLimit1.0 		:= StatusIn.2;
	Out.bLimit1.1 		:= StatusIn.3;
	Out.bLimit2.0 		:= StatusIn.4;
	Out.bLimit2.1 		:= StatusIn.5;
	Out.bError 			:= StatusIn.6;
	Out.bPDO_State 		:= StatusIn.14;
	Out.bPDO_Toggle		:= StatusIn.15;

END_FUNCTION_BLOCK

// ---- POUs/FUNCTION BLOCKS/FB_IntFilter.TcPOU
FUNCTION_BLOCK FB_IntFilter
VAR_INPUT
	ValueIn: INT := 0;
	Cycles: INT;
END_VAR
VAR_OUTPUT
	ValueOut: INT;
END_VAR
VAR
	CycleCounter: INT := 0;
	ValueSum: REAL := 0;
	ValueAverage: INT := 0;
	LoopReset: INT;
END_VAR

//CycleCounter := CycleCounter + 1;

IF CycleCounter < Cycles THEN
	ValueSum := ValueSum + INT_TO_REAL(ValueIn) ;
	CycleCounter := CycleCounter + 1;
ELSE
	ValueAverage := REAL_TO_INT(ValueSum / INT_TO_REAL(Cycles)) ;
	ValueOut := ValueAverage;
	ValueSum := 0 ;
	CycleCounter := 0 ;
END_IF

END_FUNCTION_BLOCK

// ---- POUs/MAIN FUNCTIONS/PRG_XX_Visualization_Variables.TcPOU
PROGRAM PRG_XX_Visualization_Variables
VAR
	

END_VAR

bRemote := IN_bRemote ;
bAutoCrossCutSingle := NOT IN_bAutoCrossCutDouble ;
bAutoCrossCutDouble := IN_bAutoCrossCutDouble ;
bZAxisSlow := IN_bZaxisSlow ;
bZAxisMed := NOT IN_bZaxisSlow AND NOT IN_bZaxisFast ;
bZAxisFast := IN_bZaxisFast ;
bTrtCCW := OUT_bTrtContactor AND OUT_bTrtCrgLH ;
bTrtCW := OUT_bTrtContactor AND OUT_bTrtCrgRH ;
bCrgLH := OUT_bCrgContactor AND OUT_bTrtCrgLH ;
bCrgRH := OUT_bCrgContactor AND OUT_bTrtCrgRH ;
bTeachLeft := IN_bTeachLeft ;
bTeachRight := IN_bTeachRight ;

END_PROGRAM

// ---- POUs/FUNCTION BLOCKS/InverseAnalogControl.TcPOU
FUNCTION_BLOCK InverseAnalogControl
VAR_INPUT
	
	AnalogInput			:INT; // 150 amps is the max, 32500 bit

END_VAR
VAR_OUTPUT
	
	AnalogOutput		:INT;

END_VAR
VAR

	Holder				:INT ;

END_VAR


Holder := (AnalogInput * -1) + 32767;

IF Holder < 8192 THEN
	
	AnalogOutput := 8192;
ELSE
	
	AnalogOutput := holder;
END_IF

END_FUNCTION_BLOCK

// ---- GlobalTextList.TcGTLO
TEXTLIST GlobalTextList
  721 = ''
  47 = '%.001f'
  788 = '%.01f'
  356 = '%.1f'
  64 = '%1f'
  366 = '%d'
  643 = '%i'
  230 = 'arriage LH'
  806 = 'AutoCrosscut'
  697 = 'AutoCrosscut Left'
  286 = 'AutoCrosscut Right'
  164 = 'Cable Reel'
  381 = 'Carriage'
  425 = 'Carriage LH'
  147 = 'Carriage Reference LED'
  269 = 'Carriage RH'
  759 = 'CCW'
  268 = 'Crosscut'
  957 = 'CUT'
  860 = 'CW'
  601 = 'Deg'
  712 = 'Degrees'
  377 = 'Double'
  819 = 'DOWN'
  765 = 'Drv Fwd'
  39 = 'Drv Rev'
  786 = 'Fault/Reset'
  706 = 'Field Light'
  163 = 'Horn'
  711 = 'Hose Reel'
  505 = 'Left'
  570 = 'LH'
  255 = 'Lifting Position'
  132 = 'OUT_bTurretReferenceLED'
  490 = 'Remote'
  945 = 'RETURN'
  414 = 'RH'
  577 = 'Right'
  12 = 'Saw'
  949 = 'Saw Current'
  947 = 'Single'
  274 = 'Slow / Med / Fast'
  485 = 'Sprayer'
  449 = 'Teach'
  914 = 'Travel Speed'
  265 = 'Turret Angle'
  929 = 'Turret angle'
  357 = 'Turret CCW'
  388 = 'Turret CW'
  394 = 'Turret Reference LED'
  192 = 'Turret Return'
  870 = 'UP'
  464 = 'Water Line'
  596 = 'Z-axis Speed'
END_TEXTLIST

// ---- VISUs/Visualization.TcVIS
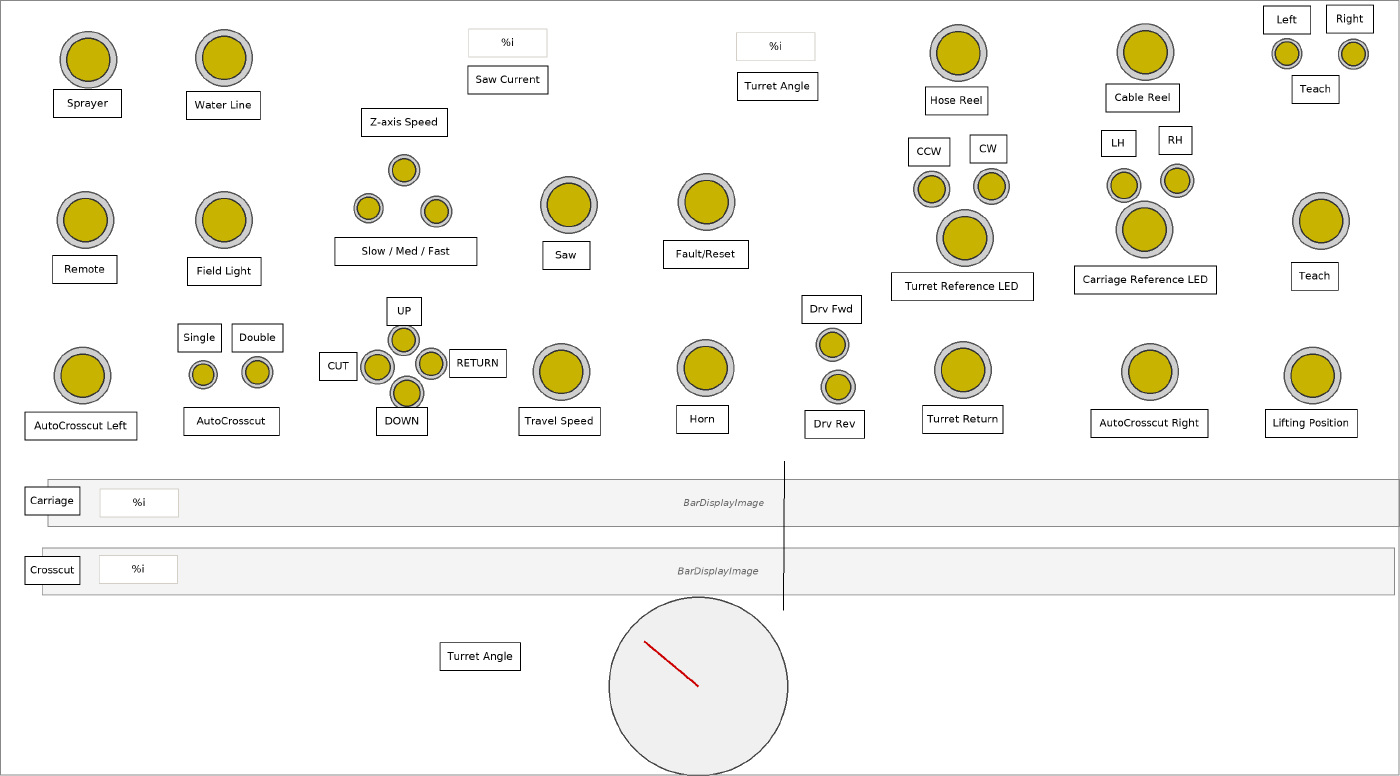
VISUALIZATION Visualization  // 1474x818
    Group (938,216 150x101)
        Lamp1 (43,0 70x70), variable: OUT_bTurretReferenceLED, style: Lamp-Lamp1-Yellow
        Rectangle (0,71 150x30), "Turret Reference LED"
    Group (1131,207 150x103)
        Lamp1 (39,0 70x70), variable: OUT_bCarriageReferenceLED, style: Lamp-Lamp1-Yellow
        Rectangle (0,73 150x30), "Carriage Reference LED"
    Lamp1 (958,177 46x45), variable: bTrtCCW, style: Lamp-Lamp1-Yellow
    Lamp1 (1020,174 48x45), variable: bTrtCW, style: Lamp-Lamp1-Yellow
    Lamp1 (1159,174 49x43), variable: bCrgLH, style: Lamp-Lamp1-Yellow
    Lamp1 (1219,170 41x41), variable: bCrgRH, style: Lamp-Lamp1-Yellow
    Rectangle (956,145 44x30), "CCW"
    Rectangle (1021,142 39x30), "CW"
    Rectangle (1159,137 37x28), "LH"
    Rectangle (1220,133 35x30), "RH"
    Lamp1 (974,21 70x70), variable: OUT_bHoseReel, style: Lamp-Lamp1-Yellow
    Lamp1 (1171,20 70x70), variable: OUT_bCableReel, style: Lamp-Lamp1-Yellow
    Lamp1 (979,355 70x70), variable: OUT_bTurretReturnLED, style: Lamp-Lamp1-Yellow
    Lamp1 (1176,357 70x70), variable: bAutoCrossCut, style: Lamp-Lamp1-Yellow
    Lamp1 (58,28 70x70), variable: OUT_bSprayer, style: Lamp-Lamp1-Yellow
    Lamp1 (201,26 70x70), variable: OUT_bWaterLine, style: Lamp-Lamp1-Yellow
    Lamp1 (55,197 70x70), variable: bRemote, style: Lamp-Lamp1-Yellow
    Lamp1 (201,197 70x70), variable: OUT_bFieldLight, style: Lamp-Lamp1-Yellow
    Lamp1 (52,361 70x70), variable: bAutoCrossCut, style: Lamp-Lamp1-Yellow
    Lamp1 (196,377 36x36), variable: bAutoCrossCutSingle, style: Lamp-Lamp1-Yellow
    Lamp1 (368,201 40x37), variable: bZAxisSlow, style: Lamp-Lamp1-Yellow
    Lamp1 (404,160 43x39), variable: bZAxisMed, style: Lamp-Lamp1-Yellow
    Lamp1 (440,203 39x40), variable: bZAxisFast, style: Lamp-Lamp1-Yellow
    Lamp1 (405,339 40x39), variable: bSawUP, style: Lamp-Lamp1-Yellow
    Lamp1 (434,364 40x39), variable: OUT_bSawRETURN, style: Lamp-Lamp1-Yellow
    Lamp1 (375,366 45x42), variable: OUT_bSawCUT, style: Lamp-Lamp1-Yellow
    Lamp1 (405,393 47x43), variable: bSawDown, style: Lamp-Lamp1-Yellow
    Lamp1 (564,181 70x70), variable: OUT_bSawONLED, style: Lamp-Lamp1-Yellow
    Lamp1 (556,357 70x70), variable: OUT_bTravelSpeedLED, style: Lamp-Lamp1-Yellow
    Lamp1 (709,178 70x70), variable: OUT_bFaultResetLED, style: Lamp-Lamp1-Yellow
    Lamp1 (708,353 70x70), variable: OUT_bHorn, style: Lamp-Lamp1-Yellow
    Lamp1 (856,343 41x41), variable: OUT_bXDriveFwd, style: Lamp-Lamp1-Yellow
    Lamp1 (857,387 51x42), variable: OUT_bXDriveRev, style: Lamp-Lamp1-Yellow
    Lamp1 (1336,37 38x39), variable: bTeachLeft, style: Lamp-Lamp1-Yellow
    Lamp1 (1402,38 46x38), variable: bTeachRight, style: Lamp-Lamp1-Yellow
    Lamp1 (1356,198 70x70), variable: OUT_bTeachLED, style: Lamp-Lamp1-Yellow
    Lamp1 (1347,361 70x70), variable: OUT_bLiftingPositionLED, style: Lamp-Lamp1-Yellow
    Rectangle (56,94 72x30), "Sprayer"
    Rectangle (196,96 78x30), "Water Line"
    Rectangle (55,269 68x30), "Remote"
    Rectangle (197,271 78x30), "Field Light"
    Rectangle (26,434 118x30), "AutoCrosscut Left"
    Rectangle (193,429 101x30), "AutoCrosscut"
    Lamp1 (251,373 40x39), variable: bAutoCrossCutDouble, style: Lamp-Lamp1-Yellow
    Rectangle (187,341 46x30), "Single"
    Rectangle (244,341 54x30), "Double"
    Rectangle (380,114 91x30), "Z-axis Speed"
    Rectangle (352,250 150x30), "Slow / Med / Fast"
    Rectangle (407,313 37x30), "UP"
    Rectangle (396,429 54x30), "DOWN"
    Rectangle (336,371 40x30), "CUT"
    Rectangle (473,368 60x30), "RETURN"
    Rectangle (571,254 50x30), "Saw"
    Rectangle (698,253 90x30), "Fault/Reset"
    Rectangle (546,429 86x30), "Travel Speed"
    Rectangle (712,427 55x30), "Horn"
    Rectangle (844,311 63x30), "Drv Fwd"
    Rectangle (847,432 63x30), "Drv Rev"
    Rectangle (971,427 85x30), "Turret Return"
    Rectangle (1148,431 124x30), "AutoCrosscut Right"
    Rectangle (974,91 66x30), "Hose Reel"
    Rectangle (1164,88 78x30), "Cable Reel"
    Rectangle (1360,79 50x30), "Teach"
    Rectangle (1359,276 50x30), "Teach"
    Rectangle (1332,431 97x30), "Lifting Position"
    Rectangle (1396,5 50x30), "Right"
    Rectangle (1330,6 50x30), "Left"
    Rectangle (776,76 85x30), "Turret Angle"
    Rectangle (492,69 85x30), "Saw Current"
    Textfield (775,34 83x30), "%i", text variable: fbTurretSSI.Out.rScaled
    Textfield (493,30 83x30), "%i", text variable: fbSawCurrent.Out.rScaled
    BarDisplayImage (50,505 1424x50), value: fbCarriagePOS.Out.rScaled, style: BarDisplayImage-Gray, scale format: %d, scale 0..41
    BarDisplayImage (44,577 1424x50), value: fbCrosscutSSI.Out.rScaled, style: BarDisplayImage-Gray, scale format: %d, scale 0..62
    Rectangle (26,513 58x30), "Carriage"
    Rectangle (26,586 58x30), "Crosscut"
    Textfield (105,515 83x30), "%i", text variable: fbCarriagePOS.Out.rScaled
    Textfield (104,585 83x30), "%i", text variable: fbCrosscutSSI.Out.rScaled
    Meter180 (552,629 366x189), value: fbTurretSSI.Out.rScaled, style: Meter-Meter180-Gray, scale format: %d, scale -90..90
        p518627256: Turret angle
    Rectangle (463,677 85x30), "Turret Angle"
    Line (825,643) (826,486)
END_VISUALIZATION
